// TIA Portal project "ConectaTwo" (V16)

(* hardware
DEVICE "S71500/ET200MP station_1"  S7-1500 station
   slot 0: "Rail_0"  Rack  6ES7 590-1***0-0AA0
   slot 1: "PLC_1"  CPU 1516-3 PN/DP  6ES7 516-3AN00-0AB0  V1.8
      slot 3: "CPU display_1"  6ES7591-1BA00-0AA0
      slot 32768: "PROFINET interface_1"  X1
         slot 32769: "Port_1"  X1 P1
         slot 32770: "Port_2"  X1 P2
      slot 33024: "PROFINET interface_2"  X2
         slot 33025: "Port_1"  X2 P1
      slot 33280: "DP interface_1"  X3
DEVICE "S71500/ET200MP station_2"  S7-1500 station
   slot 0: "Rail_0"  Rack  6ES7 590-1***0-0AA0
   slot 1: "PLC_2"  CPU 1516-3 PN/DP  6ES7 516-3AN00-0AB0  V1.8
      slot 3: "CPU display_1"  6ES7591-1BA00-0AA0
      slot 32768: "PROFINET interface_1"  X1
         slot 32769: "Port_1"  X1 P1
         slot 32770: "Port_2"  X1 P2
      slot 33024: "PROFINET interface_2"  X2
         slot 33025: "Port_1"  X2 P1
      slot 33280: "DP interface_1"  X3
DEVICE "HMI_1"  TP700 Comfort
   slot 0: "HMI_1"  TP700 Comfort  6AV2 124-0GC01-0AX0  16.0.0.0
   slot 1: "HMI_RT_1"  TP700 Comfort  6AV2 124-0GC01-0AX0  16.0.0.0
   slot 5: "HMI_1.IE_CP_1"  PROFINET Interface  16.0.0.0
      slot 1: "PROFINET Interface_1"  PROFINET Interface
         slot 1: "Port_1"  Port
         slot 2: "Port_2"  Port
   slot 7: "HMI_1.MPI/DP_CP_1"  MPI/DP Interface  16.0.0.0
DEVICE "HMI_2"  TP700 Comfort
   slot 0: "HMI_2"  TP700 Comfort  6AV2 124-0GC01-0AX0  16.0.0.0
   slot 1: "HMI_RT_2"  TP700 Comfort  6AV2 124-0GC01-0AX0  16.0.0.0
   slot 5: "HMI_2.IE_CP_1"  PROFINET Interface  16.0.0.0
      slot 1: "PROFINET Interface_1"  PROFINET Interface
         slot 1: "Port_1"  Port
         slot 2: "Port_2"  Port
   slot 7: "HMI_2.MPI/DP_CP_1"  MPI/DP Interface  16.0.0.0
*)

// ===== PLC "PLC_1"  CPU 1516-3 PN/DP =====

VAR_GLOBAL   // PLC tag table "Default tag table"
   "Clock_Byte" AT %MB10 : Byte;
   "Clock_10Hz" AT %M10.0 : Bool;
   "Clock_1Hz" AT %M10.5 : Bool;
   "Mensaje1J1" AT %M11.0 : Bool;
   "Mensaje2J1" AT %M11.1 : Bool;
   "Mensaje3J1" AT %M11.2 : Bool;
   "Mensaje4J1" AT %M11.3 : Bool;
   "Mensaje5J1" AT %M11.4 : Bool;
   "Mensaje6J1" AT %M11.5 : Bool;
   "Mensaje7J1" AT %M11.6 : Bool;
   "B1J1" AT %M11.7 : Bool;
   "B2J1" AT %M12.0 : Bool;
   "B3J1" AT %M12.1 : Bool;
   "B4J1" AT %M12.2 : Bool;
   "B5J1" AT %M12.3 : Bool;
   "B6J1" AT %M12.4 : Bool;
   "B7J1" AT %M12.5 : Bool;
   "B8J1" AT %M12.6 : Bool;
   "B9J1" AT %M12.7 : Bool;
   "PanelJ1" AT %M13.0 : Bool;
   "ReiniciarJ1" AT %M13.1 : Bool;
   "Conecta4J1" AT %M13.2 : Bool;
   "Conecta5J1" AT %M13.3 : Bool;
   "Conecta4SJ1" AT %M13.4 : Bool;
   "Conecta5SJ1" AT %M13.5 : Bool;
   "ModoJuegoJ1Send" AT %MW14 : Int;
   "ModoJuegoJ2Rec" AT %MW16 : Int;
   "ResetJ1Send" AT %M18.0 : Bool;
   "ResetJ2Rec" AT %M18.1 : Bool;
   "EstadoTurnoAJ1Send" AT %M18.2 : Bool;
   "EstadoTurnoAJ2Rec" AT %M18.3 : Bool;
   "EstadoTurnoBJ1Send" AT %M18.4 : Bool;
   "EstadoTurnoBJ2Rec" AT %M18.5 : Bool;
   "CambioBJ1" AT %M18.6 : Bool;
   "CambioVectorJ1" AT %M18.7 : Bool;
END_VAR

DATA_BLOCK "Jugador1Vect"   // DB4
{ S7_Optimized_Access := 'FALSE' }
VERSION : 0.1
   VAR
      J1Vect : Array[0..7, 0..8] of Int;
      J1VecSend : Array[0..7, 0..8] of Int;
      J1VecRec : Array[0..7, 0..8] of Int;
   END_VAR
BEGIN
   J1Vect[0,0] := 0;
   J1Vect[0,1] := 0;
   J1Vect[0,2] := 0;
   J1Vect[0,3] := 0;
   J1Vect[0,4] := 0;
   J1Vect[0,6] := 0;
   J1Vect[0,7] := 0;
   J1Vect[0,8] := 0;
   J1Vect[1,0] := 0;
   J1Vect[1,1] := 0;
   J1Vect[1,3] := 0;
   J1VecSend[1,3] := 0;
   J1VecSend[1,1] := 0;
   J1VecSend[1,0] := 0;
   J1VecSend[0,8] := 0;
   J1VecSend[0,7] := 0;
   J1VecSend[0,6] := 0;
   J1VecSend[0,4] := 0;
   J1VecSend[0,3] := 0;
   J1VecSend[0,2] := 0;
   J1VecSend[0,1] := 0;
   J1VecSend[0,0] := 0;
   J1VecRec[0,0] := 0;
   J1VecRec[0,1] := 0;
   J1VecRec[0,2] := 0;
   J1VecRec[0,3] := 0;
   J1VecRec[0,4] := 0;
   J1VecRec[0,6] := 0;
   J1VecRec[0,7] := 0;
   J1VecRec[0,8] := 0;
   J1VecRec[1,0] := 0;
   J1VecRec[1,1] := 0;
   J1VecRec[1,3] := 0;
END_DATA_BLOCK

// folder: System blocks/Program resources

DATA_BLOCK "EnviarModo"   // DB3
{ S7_Optimized_Access := 'TRUE' }
AUTHOR : SIMATIC
FAMILY : MC7Plus
NAME : TC_IP_v4
VERSION : 1.0
// stored: InstanceOfName TCON_IP_v4
"TCON_IP_v4"
BEGIN
   ID := 1;
   InterfaceId := 64;
   RemotePort := 2000;
   ActiveEstablished := true;
   RemoteAddress.ADDR[1] := 192;
   RemoteAddress.ADDR[2] := 168;
   RemoteAddress.ADDR[3] := 50;
   RemoteAddress.ADDR[4] := 2;
END_DATA_BLOCK

DATA_BLOCK "EnviarReset"   // DB6
{ S7_Optimized_Access := 'TRUE' }
AUTHOR : SIMATIC
FAMILY : MC7Plus
NAME : TC_IP_v4
VERSION : 1.0
// stored: InstanceOfName TCON_IP_v4
"TCON_IP_v4"
BEGIN
   ID := 2;
   InterfaceId := 64;
   RemotePort := 2010;
   ActiveEstablished := true;
   RemoteAddress.ADDR[1] := 192;
   RemoteAddress.ADDR[2] := 168;
   RemoteAddress.ADDR[3] := 50;
   RemoteAddress.ADDR[4] := 2;
END_DATA_BLOCK

DATA_BLOCK "EnviarTurnoA"   // DB7
{ S7_Optimized_Access := 'TRUE' }
AUTHOR : SIMATIC
FAMILY : MC7Plus
NAME : TC_IP_v4
VERSION : 1.0
// stored: InstanceOfName TCON_IP_v4
"TCON_IP_v4"
BEGIN
   ID := 3;
   InterfaceId := 64;
   RemotePort := 2020;
   ActiveEstablished := true;
   RemoteAddress.ADDR[1] := 192;
   RemoteAddress.ADDR[2] := 168;
   RemoteAddress.ADDR[3] := 50;
   RemoteAddress.ADDR[4] := 2;
END_DATA_BLOCK

DATA_BLOCK "RecibirTurnoB"   // DB9
{ S7_Optimized_Access := 'TRUE' }
AUTHOR : SIMATIC
FAMILY : MC7Plus
NAME : TC_IP_v4
VERSION : 1.0
// stored: InstanceOfName TCON_IP_v4
"TCON_IP_v4"
BEGIN
   ID := 4;
   InterfaceId := 64;
   LocalPort := 2030;
   RemoteAddress.ADDR[1] := 192;
   RemoteAddress.ADDR[2] := 168;
   RemoteAddress.ADDR[3] := 50;
   RemoteAddress.ADDR[4] := 2;
END_DATA_BLOCK

DATA_BLOCK "EnviarVectorA"   // DB12
{ S7_Optimized_Access := 'TRUE' }
AUTHOR : SIMATIC
FAMILY : MC7Plus
NAME : TC_IP_v4
VERSION : 1.0
// stored: InstanceOfName TCON_IP_v4
"TCON_IP_v4"
BEGIN
   ID := 5;
   InterfaceId := 64;
   RemotePort := 2040;
   ActiveEstablished := true;
   RemoteAddress.ADDR[1] := 192;
   RemoteAddress.ADDR[2] := 168;
   RemoteAddress.ADDR[3] := 50;
   RemoteAddress.ADDR[4] := 2;
END_DATA_BLOCK

DATA_BLOCK "RecibirVectorB"   // DB13
{ S7_Optimized_Access := 'TRUE' }
AUTHOR : SIMATIC
FAMILY : MC7Plus
NAME : TC_IP_v4
VERSION : 1.0
// stored: InstanceOfName TCON_IP_v4
"TCON_IP_v4"
BEGIN
   ID := 6;
   InterfaceId := 64;
   LocalPort := 2050;
   RemoteAddress.ADDR[1] := 192;
   RemoteAddress.ADDR[2] := 168;
   RemoteAddress.ADDR[3] := 50;
   RemoteAddress.ADDR[4] := 2;
END_DATA_BLOCK

// folder: (top level)

ORGANIZATION_BLOCK "Main"   // OB1, LAD, ProgramCycle
TITLE = "Main Program Sweep (Cycle)"
{ S7_Optimized_Access := 'TRUE' }
VERSION : 0.1
   VAR_INPUT
      Initial_Call : Bool;   // Initial call of this OB
      Remanence : Bool;   // =True, if remanent data are available
   END_VAR
BEGIN

REGION Network 1: Enviar y Recibir Modo de Juego
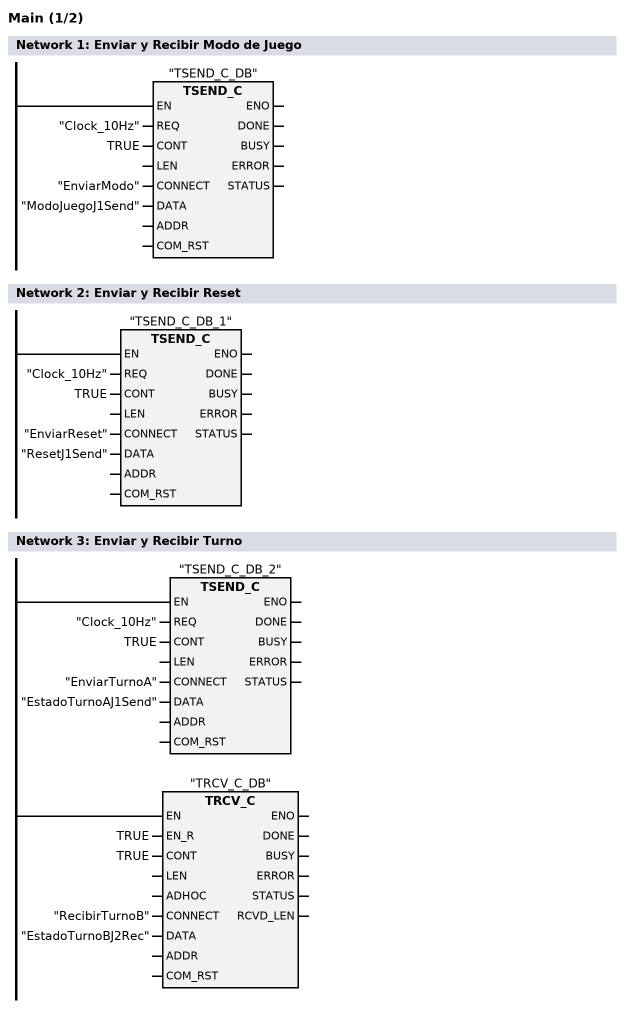
   "TSEND_C_DB"(REQ := "Clock_10Hz", CONT := TRUE, CONNECT := "EnviarModo", DATA := "ModoJuegoJ1Send");   // TSEND_C
END_REGION

REGION Network 2: Enviar y Recibir Reset
   "TSEND_C_DB_1"(REQ := "Clock_10Hz", CONT := TRUE, CONNECT := "EnviarReset", DATA := "ResetJ1Send");   // TSEND_C
END_REGION

REGION Network 3: Enviar y Recibir Turno
   "TSEND_C_DB_2"(REQ := "Clock_10Hz", CONT := TRUE, CONNECT := "EnviarTurnoA", DATA := "EstadoTurnoAJ1Send");   // TSEND_C
   "TRCV_C_DB"(EN_R := TRUE, CONT := TRUE, CONNECT := "RecibirTurnoB", DATA := "EstadoTurnoBJ2Rec");   // TRCV_C
END_REGION

REGION Network 4: Enviar y Recibir Vector
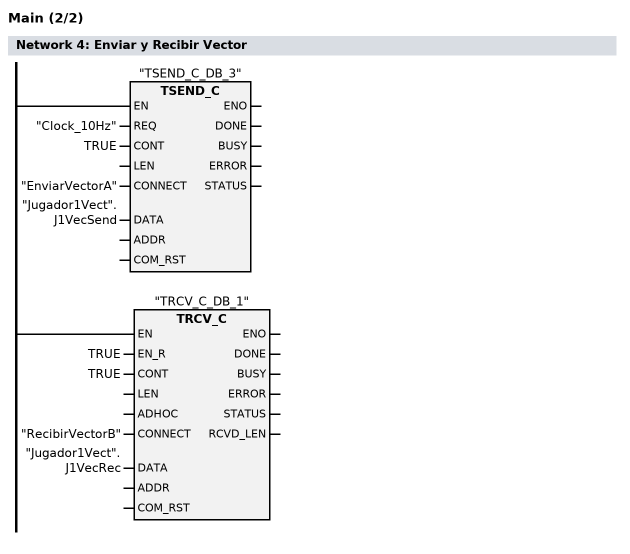
   "TSEND_C_DB_3"(REQ := "Clock_10Hz",   // TSEND_C
                  CONT := TRUE,
                  CONNECT := "EnviarVectorA",
                  DATA := "Jugador1Vect".J1VecSend);
   "TRCV_C_DB_1"(EN_R := TRUE, CONT := TRUE, CONNECT := "RecibirVectorB", DATA := "Jugador1Vect".J1VecRec);   // TRCV_C
END_REGION

REGION Network 5 (SCL): Checar si ganador rojo
   IF "ReiniciarJ1" = TRUE THEN
       "ResetJ1Send" := TRUE;
       "ModoJuegoJ1Send" := 0;
       "ModoJuegoJ2Rec" := 0;
       FILL_BLK(IN:=0,
                COUNT:=72,
                OUT=>"Jugador1Vect".J1Vect[0,0]);
       FILL_BLK(IN := 0,
                COUNT := 72,
                OUT => "Jugador1Vect".J1VecSend[0, 0]);
       FILL_BLK(IN := 0,
                COUNT := 72,
                OUT => "Jugador1Vect".J1VecRec[0, 0]);
       "Mensaje1J1" := FALSE;
       "Mensaje2J1" := FALSE;
       "Mensaje3J1" := FALSE;
       "Mensaje4J1" := FALSE;
       "Mensaje5J1" := FALSE;
       "Mensaje6J1" := FALSE;
       "Mensaje7J1" := FALSE;
       "EstadoTurnoAJ1Send" := TRUE;
       "EstadoTurnoAJ2Rec" := FALSE;
       "EstadoTurnoBJ1Send" := FALSE;
       "EstadoTurnoBJ2Rec" := FALSE;
       "Conecta4SJ1" := FALSE;
       "Conecta5SJ1" := FALSE;
       "PanelJ1" := FALSE;
       "CambioBJ1" := FALSE;
       "CambioVectorJ1" := FALSE;
   ELSE
       "ResetJ1Send" := FALSE;
   END_IF;

   IF "ModoJuegoJ1Send" = 0 THEN
       IF "Conecta4J1" = TRUE THEN
           "Conecta4SJ1" := TRUE;
           "ModoJuegoJ1Send" := 4;
           "Mensaje1J1" := TRUE;
           "Mensaje2J1" := TRUE;
           "Mensaje3J1" := FALSE;
       END_IF;
       IF "Conecta5J1" = TRUE THEN
           "Conecta5SJ1" := TRUE;
           "ModoJuegoJ1Send" := 5;
           "Mensaje1J1" := TRUE;
           "Mensaje3J1" := TRUE;
           "Mensaje2J1" := FALSE;
       END_IF;
   END_IF;

   IF "Conecta4SJ1" = TRUE OR "Conecta5SJ1" = TRUE THEN
       IF "EstadoTurnoAJ1Send" = TRUE THEN
           "PanelJ1" := TRUE;
           "Mensaje4J1" := TRUE;
           "Mensaje5J1" := FALSE;
       ELSE
           "PanelJ1" := FALSE;
           "Mensaje4J1" := FALSE;
           "Mensaje5J1" := TRUE;
       END_IF;
   END_IF;

   IF "B1J1" OR "B2J1" OR "B3J1" OR "B4J1" OR "B5J1" OR "B6J1" OR "B7J1" OR "B7J1" OR "B8J1" OR "B9J1" OR "EstadoTurnoBJ2Rec" THEN
       IF "EstadoTurnoAJ1Send" = TRUE THEN
           "EstadoTurnoAJ1Send" := FALSE;
       ELSE
           "EstadoTurnoAJ1Send" := TRUE;
       END_IF;
   END_IF;

   IF "B1J1" AND "CambioBJ1" = FALSE THEN
       MOVE_BLK(IN := "Jugador1Vect".J1VecRec[0, 0],
                COUNT := 72,
                OUT => "Jugador1Vect".J1Vect[0, 0]);
       IF "Jugador1Vect".J1Vect[0, 0] = 0 THEN
           "Jugador1Vect".J1Vect[0, 0] := 2;
           "CambioBJ1" := TRUE;
           MOVE_BLK(IN := "Jugador1Vect".J1Vect[0, 0],
                    COUNT := 72,
                    OUT => "Jugador1Vect".J1VecSend[0, 0]);
       ELSIF "Jugador1Vect".J1Vect[1, 0] = 0 THEN
           "Jugador1Vect".J1Vect[1, 0] := 2;
           "CambioBJ1" := TRUE;
           MOVE_BLK(IN := "Jugador1Vect".J1VecRec[0, 0],
                    COUNT := 72,
                    OUT => "Jugador1Vect".J1Vect[0, 0]);
       ELSIF "Jugador1Vect".J1Vect[2, 0] = 0 THEN
           "Jugador1Vect".J1Vect[2, 0] := 2;
           "CambioBJ1" := TRUE;
           MOVE_BLK(IN := "Jugador1Vect".J1Vect[0, 0],
                    COUNT := 72,
                    OUT => "Jugador1Vect".J1VecSend[0, 0]);
       ELSIF "Jugador1Vect".J1Vect[3, 0] = 0 THEN
           "Jugador1Vect".J1Vect[3, 0] := 2;
           "CambioBJ1" := TRUE;
           MOVE_BLK(IN := "Jugador1Vect".J1VecRec[0, 0],
                    COUNT := 72,
                    OUT => "Jugador1Vect".J1Vect[0, 0]);
       ELSIF "Jugador1Vect".J1Vect[4, 0] = 0 THEN
           "Jugador1Vect".J1Vect[4, 0] := 2;
           "CambioBJ1" := TRUE;
           MOVE_BLK(IN := "Jugador1Vect".J1Vect[0, 0],
                    COUNT := 72,
                    OUT => "Jugador1Vect".J1VecSend[0, 0]);
       ELSIF "Jugador1Vect".J1Vect[5, 0] = 0 THEN
           "Jugador1Vect".J1Vect[5, 0] := 2;
           "CambioBJ1" := TRUE;
           MOVE_BLK(IN := "Jugador1Vect".J1Vect[0, 0],
                    COUNT := 72,
                    OUT => "Jugador1Vect".J1VecSend[0, 0]);
       ELSIF "Jugador1Vect".J1Vect[6, 0] = 0 THEN
           "Jugador1Vect".J1Vect[6, 0] := 2;
           "CambioBJ1" := TRUE;
           MOVE_BLK(IN := "Jugador1Vect".J1Vect[0, 0],
                    COUNT := 72,
                    OUT => "Jugador1Vect".J1VecSend[0, 0]);
       ELSIF "Jugador1Vect".J1Vect[7, 0] = 0 THEN
           "Jugador1Vect".J1Vect[7, 0] := 2;
           "CambioBJ1" := TRUE;
           MOVE_BLK(IN := "Jugador1Vect".J1Vect[0, 0],
                    COUNT := 72,
                    OUT => "Jugador1Vect".J1VecSend[0, 0]);
       END_IF;
   END_IF;

   IF "B2J1" AND "CambioBJ1" = FALSE THEN
       MOVE_BLK(IN := "Jugador1Vect".J1VecRec[0, 0],
                COUNT := 72,
                OUT => "Jugador1Vect".J1Vect[0, 0]);
       IF "Jugador1Vect".J1Vect[0, 1] = 0 THEN
           "Jugador1Vect".J1Vect[0, 1] := 2;
           "CambioBJ1" := TRUE;
           MOVE_BLK(IN := "Jugador1Vect".J1Vect[0, 0],
                    COUNT := 72,
                    OUT => "Jugador1Vect".J1VecSend[0, 0]);
       ELSIF "Jugador1Vect".J1Vect[1, 1] = 0 THEN
           "Jugador1Vect".J1Vect[1, 1] := 2;
           "CambioBJ1" := TRUE;
           MOVE_BLK(IN := "Jugador1Vect".J1VecRec[0, 0],
                    COUNT := 72,
                    OUT => "Jugador1Vect".J1Vect[0, 0]);
       ELSIF "Jugador1Vect".J1Vect[2, 1] = 0 THEN
           "Jugador1Vect".J1Vect[2, 1] := 2;
           "CambioBJ1" := TRUE;
           MOVE_BLK(IN := "Jugador1Vect".J1Vect[0, 0],
                    COUNT := 72,
                    OUT => "Jugador1Vect".J1VecSend[0, 0]);
       ELSIF "Jugador1Vect".J1Vect[3, 1] = 0 THEN
           "Jugador1Vect".J1Vect[3, 1] := 2;
           "CambioBJ1" := TRUE;
           MOVE_BLK(IN := "Jugador1Vect".J1VecRec[0, 0],
                    COUNT := 72,
                    OUT => "Jugador1Vect".J1Vect[0, 0]);
       ELSIF "Jugador1Vect".J1Vect[4, 1] = 0 THEN
           "Jugador1Vect".J1Vect[4, 1] := 2;
           "CambioBJ1" := TRUE;
           MOVE_BLK(IN := "Jugador1Vect".J1Vect[0, 0],
                    COUNT := 72,
                    OUT => "Jugador1Vect".J1VecSend[0, 0]);
       ELSIF "Jugador1Vect".J1Vect[5, 1] = 0 THEN
           "Jugador1Vect".J1Vect[5, 1] := 2;
           "CambioBJ1" := TRUE;
           MOVE_BLK(IN := "Jugador1Vect".J1Vect[0, 0],
                    COUNT := 72,
                    OUT => "Jugador1Vect".J1VecSend[0, 0]);
       ELSIF "Jugador1Vect".J1Vect[6, 1] = 0 THEN
           "Jugador1Vect".J1Vect[6, 1] := 2;
           "CambioBJ1" := TRUE;
           MOVE_BLK(IN := "Jugador1Vect".J1Vect[0, 0],
                    COUNT := 72,
                    OUT => "Jugador1Vect".J1VecSend[0, 0]);
       ELSIF "Jugador1Vect".J1Vect[7, 1] = 0 THEN
           "Jugador1Vect".J1Vect[7, 1] := 2;
           "CambioBJ1" := TRUE;
           MOVE_BLK(IN := "Jugador1Vect".J1Vect[0, 0],
                    COUNT := 72,
                    OUT => "Jugador1Vect".J1VecSend[0, 0]);
       END_IF;
   END_IF;

   IF "B3J1" AND "CambioBJ1" = FALSE THEN
       MOVE_BLK(IN := "Jugador1Vect".J1VecRec[0, 0],
                COUNT := 72,
                OUT => "Jugador1Vect".J1Vect[0, 0]);
       IF "Jugador1Vect".J1Vect[0, 2] = 0 THEN
           "Jugador1Vect".J1Vect[0, 2] := 2;
           "CambioBJ1" := TRUE;
           MOVE_BLK(IN := "Jugador1Vect".J1Vect[0, 0],
                    COUNT := 72,
                    OUT => "Jugador1Vect".J1VecSend[0, 0]);
       ELSIF "Jugador1Vect".J1Vect[1, 2] = 0 THEN
           "Jugador1Vect".J1Vect[1, 2] := 2;
           "CambioBJ1" := TRUE;
           MOVE_BLK(IN := "Jugador1Vect".J1VecRec[0, 0],
                    COUNT := 72,
                    OUT => "Jugador1Vect".J1Vect[0, 0]);
       ELSIF "Jugador1Vect".J1Vect[2, 2] = 0 THEN
           "Jugador1Vect".J1Vect[2, 2] := 2;
           "CambioBJ1" := TRUE;
           MOVE_BLK(IN := "Jugador1Vect".J1Vect[0, 0],
                    COUNT := 72,
                    OUT => "Jugador1Vect".J1VecSend[0, 0]);
       ELSIF "Jugador1Vect".J1Vect[3, 2] = 0 THEN
           "Jugador1Vect".J1Vect[3, 2] := 2;
           "CambioBJ1" := TRUE;
           MOVE_BLK(IN := "Jugador1Vect".J1VecRec[0, 0],
                    COUNT := 72,
                    OUT => "Jugador1Vect".J1Vect[0, 0]);
       ELSIF "Jugador1Vect".J1Vect[4, 2] = 0 THEN
           "Jugador1Vect".J1Vect[4, 2] := 2;
           "CambioBJ1" := TRUE;
           MOVE_BLK(IN := "Jugador1Vect".J1Vect[0, 0],
                    COUNT := 72,
                    OUT => "Jugador1Vect".J1VecSend[0, 0]);
       ELSIF "Jugador1Vect".J1Vect[5, 2] = 0 THEN
           "Jugador1Vect".J1Vect[5, 2] := 2;
           "CambioBJ1" := TRUE;
           MOVE_BLK(IN := "Jugador1Vect".J1Vect[0, 0],
                    COUNT := 72,
                    OUT => "Jugador1Vect".J1VecSend[0, 0]);
       ELSIF "Jugador1Vect".J1Vect[6, 2] = 0 THEN
           "Jugador1Vect".J1Vect[6, 2] := 2;
           "CambioBJ1" := TRUE;
           MOVE_BLK(IN := "Jugador1Vect".J1Vect[0, 0],
                    COUNT := 72,
                    OUT => "Jugador1Vect".J1VecSend[0, 0]);
       ELSIF "Jugador1Vect".J1Vect[7, 2] = 0 THEN
           "Jugador1Vect".J1Vect[7, 2] := 2;
           "CambioBJ1" := TRUE;
           MOVE_BLK(IN := "Jugador1Vect".J1Vect[0, 0],
                    COUNT := 72,
                    OUT => "Jugador1Vect".J1VecSend[0, 0]);
       END_IF;
   END_IF;

   IF "B4J1" AND "CambioBJ1" = FALSE THEN
       MOVE_BLK(IN := "Jugador1Vect".J1VecRec[0, 0],
                COUNT := 72,
                OUT => "Jugador1Vect".J1Vect[0, 0]);
       IF "Jugador1Vect".J1Vect[0, 3] = 0 THEN
           "Jugador1Vect".J1Vect[0, 3] := 2;
           "CambioBJ1" := TRUE;
           MOVE_BLK(IN := "Jugador1Vect".J1Vect[0, 0],
                    COUNT := 72,
                    OUT => "Jugador1Vect".J1VecSend[0, 0]);
       ELSIF "Jugador1Vect".J1Vect[1, 3] = 0 THEN
           "Jugador1Vect".J1Vect[1, 3] := 2;
           "CambioBJ1" := TRUE;
           MOVE_BLK(IN := "Jugador1Vect".J1VecRec[0, 0],
                    COUNT := 72,
                    OUT => "Jugador1Vect".J1Vect[0, 0]);
       ELSIF "Jugador1Vect".J1Vect[2, 3] = 0 THEN
           "Jugador1Vect".J1Vect[2, 3] := 2;
           "CambioBJ1" := TRUE;
           MOVE_BLK(IN := "Jugador1Vect".J1Vect[0, 0],
                    COUNT := 72,
                    OUT => "Jugador1Vect".J1VecSend[0, 0]);
       ELSIF "Jugador1Vect".J1Vect[3, 3] = 0 THEN
           "Jugador1Vect".J1Vect[3, 3] := 2;
           "CambioBJ1" := TRUE;
           MOVE_BLK(IN := "Jugador1Vect".J1VecRec[0, 0],
                    COUNT := 72,
                    OUT => "Jugador1Vect".J1Vect[0, 0]);
       ELSIF "Jugador1Vect".J1Vect[4, 3] = 0 THEN
           "Jugador1Vect".J1Vect[4, 3] := 2;
           "CambioBJ1" := TRUE;
           MOVE_BLK(IN := "Jugador1Vect".J1Vect[0, 0],
                    COUNT := 72,
                    OUT => "Jugador1Vect".J1VecSend[0, 0]);
       ELSIF "Jugador1Vect".J1Vect[5, 3] = 0 THEN
           "Jugador1Vect".J1Vect[5, 3] := 2;
           "CambioBJ1" := TRUE;
           MOVE_BLK(IN := "Jugador1Vect".J1Vect[0, 0],
                    COUNT := 72,
                    OUT => "Jugador1Vect".J1VecSend[0, 0]);
       ELSIF "Jugador1Vect".J1Vect[6, 3] = 0 THEN
           "Jugador1Vect".J1Vect[6, 3] := 2;
           "CambioBJ1" := TRUE;
           MOVE_BLK(IN := "Jugador1Vect".J1Vect[0, 0],
                    COUNT := 72,
                    OUT => "Jugador1Vect".J1VecSend[0, 0]);
       ELSIF "Jugador1Vect".J1Vect[7, 3] = 0 THEN
           "Jugador1Vect".J1Vect[7, 3] := 2;
           "CambioBJ1" := TRUE;
           MOVE_BLK(IN := "Jugador1Vect".J1Vect[0, 0],
                    COUNT := 72,
                    OUT => "Jugador1Vect".J1VecSend[0, 0]);
       END_IF;
   END_IF;

   IF "B5J1" AND "CambioBJ1" = FALSE THEN
       MOVE_BLK(IN := "Jugador1Vect".J1VecRec[0, 0],
                COUNT := 72,
                OUT => "Jugador1Vect".J1Vect[0, 0]);
       IF "Jugador1Vect".J1Vect[0, 4] = 0 THEN
           "Jugador1Vect".J1Vect[0, 4] := 2;
           "CambioBJ1" := TRUE;
           MOVE_BLK(IN := "Jugador1Vect".J1Vect[0, 0],
                    COUNT := 72,
                    OUT => "Jugador1Vect".J1VecSend[0, 0]);
       ELSIF "Jugador1Vect".J1Vect[1, 4] = 0 THEN
           "Jugador1Vect".J1Vect[1, 4] := 2;
           "CambioBJ1" := TRUE;
           MOVE_BLK(IN := "Jugador1Vect".J1VecRec[0, 0],
                    COUNT := 72,
                    OUT => "Jugador1Vect".J1Vect[0, 0]);
       ELSIF "Jugador1Vect".J1Vect[2, 4] = 0 THEN
           "Jugador1Vect".J1Vect[2, 4] := 2;
           "CambioBJ1" := TRUE;
           MOVE_BLK(IN := "Jugador1Vect".J1Vect[0, 0],
                    COUNT := 72,
                    OUT => "Jugador1Vect".J1VecSend[0, 0]);
       ELSIF "Jugador1Vect".J1Vect[3, 4] = 0 THEN
           "Jugador1Vect".J1Vect[3, 4] := 2;
           "CambioBJ1" := TRUE;
           MOVE_BLK(IN := "Jugador1Vect".J1VecRec[0, 0],
                    COUNT := 72,
                    OUT => "Jugador1Vect".J1Vect[0, 0]);
       ELSIF "Jugador1Vect".J1Vect[4, 4] = 0 THEN
           "Jugador1Vect".J1Vect[4, 4] := 2;
           "CambioBJ1" := TRUE;
           MOVE_BLK(IN := "Jugador1Vect".J1Vect[0, 0],
                    COUNT := 72,
                    OUT => "Jugador1Vect".J1VecSend[0, 0]);
       ELSIF "Jugador1Vect".J1Vect[5, 4] = 0 THEN
           "Jugador1Vect".J1Vect[5, 4] := 2;
           "CambioBJ1" := TRUE;
           MOVE_BLK(IN := "Jugador1Vect".J1Vect[0, 0],
                    COUNT := 72,
                    OUT => "Jugador1Vect".J1VecSend[0, 0]);
       ELSIF "Jugador1Vect".J1Vect[6, 4] = 0 THEN
           "Jugador1Vect".J1Vect[6, 4] := 2;
           "CambioBJ1" := TRUE;
           MOVE_BLK(IN := "Jugador1Vect".J1Vect[0, 0],
                    COUNT := 72,
                    OUT => "Jugador1Vect".J1VecSend[0, 0]);
       ELSIF "Jugador1Vect".J1Vect[7, 4] = 0 THEN
           "Jugador1Vect".J1Vect[7, 4] := 2;
           "CambioBJ1" := TRUE;
           MOVE_BLK(IN := "Jugador1Vect".J1Vect[0, 0],
                    COUNT := 72,
                    OUT => "Jugador1Vect".J1VecSend[0, 0]);
       END_IF;
   END_IF;

   IF "B6J1" AND "CambioBJ1" = FALSE THEN
       MOVE_BLK(IN := "Jugador1Vect".J1VecRec[0, 0],
                COUNT := 72,
                OUT => "Jugador1Vect".J1Vect[0, 0]);
       IF "Jugador1Vect".J1Vect[0, 5] = 0 THEN
           "Jugador1Vect".J1Vect[0, 5] := 2;
           "CambioBJ1" := TRUE;
           MOVE_BLK(IN := "Jugador1Vect".J1Vect[0, 0],
                    COUNT := 72,
                    OUT => "Jugador1Vect".J1VecSend[0, 0]);
       ELSIF "Jugador1Vect".J1Vect[1, 5] = 0 THEN
           "Jugador1Vect".J1Vect[1, 5] := 2;
           "CambioBJ1" := TRUE;
           MOVE_BLK(IN := "Jugador1Vect".J1VecRec[0, 0],
                    COUNT := 72,
                    OUT => "Jugador1Vect".J1Vect[0, 0]);
       ELSIF "Jugador1Vect".J1Vect[2, 5] = 0 THEN
           "Jugador1Vect".J1Vect[2, 5] := 2;
           "CambioBJ1" := TRUE;
           MOVE_BLK(IN := "Jugador1Vect".J1Vect[0, 0],
                    COUNT := 72,
                    OUT => "Jugador1Vect".J1VecSend[0, 0]);
       ELSIF "Jugador1Vect".J1Vect[3, 5] = 0 THEN
           "Jugador1Vect".J1Vect[3, 5] := 2;
           "CambioBJ1" := TRUE;
           MOVE_BLK(IN := "Jugador1Vect".J1VecRec[0, 0],
                    COUNT := 72,
                    OUT => "Jugador1Vect".J1Vect[0, 0]);
       ELSIF "Jugador1Vect".J1Vect[4, 5] = 0 THEN
           "Jugador1Vect".J1Vect[4, 5] := 2;
           "CambioBJ1" := TRUE;
           MOVE_BLK(IN := "Jugador1Vect".J1Vect[0, 0],
                    COUNT := 72,
                    OUT => "Jugador1Vect".J1VecSend[0, 0]);
       ELSIF "Jugador1Vect".J1Vect[5, 5] = 0 THEN
           "Jugador1Vect".J1Vect[5, 5] := 2;
           "CambioBJ1" := TRUE;
           MOVE_BLK(IN := "Jugador1Vect".J1Vect[0, 0],
                    COUNT := 72,
                    OUT => "Jugador1Vect".J1VecSend[0, 0]);
       ELSIF "Jugador1Vect".J1Vect[6, 5] = 0 THEN
           "Jugador1Vect".J1Vect[6, 5] := 2;
           "CambioBJ1" := TRUE;
           MOVE_BLK(IN := "Jugador1Vect".J1Vect[0, 0],
                    COUNT := 72,
                    OUT => "Jugador1Vect".J1VecSend[0, 0]);
       ELSIF "Jugador1Vect".J1Vect[7, 5] = 0 THEN
           "Jugador1Vect".J1Vect[7, 5] := 2;
           "CambioBJ1" := TRUE;
           MOVE_BLK(IN := "Jugador1Vect".J1Vect[0, 0],
                    COUNT := 72,
                    OUT => "Jugador1Vect".J1VecSend[0, 0]);
       END_IF;
   END_IF;

   IF "B7J1" AND "CambioBJ1" = FALSE THEN
       MOVE_BLK(IN := "Jugador1Vect".J1VecRec[0, 0],
                COUNT := 72,
                OUT => "Jugador1Vect".J1Vect[0, 0]);
       IF "Jugador1Vect".J1Vect[0, 6] = 0 THEN
           "Jugador1Vect".J1Vect[0, 6] := 2;
           "CambioBJ1" := TRUE;
           MOVE_BLK(IN := "Jugador1Vect".J1Vect[0, 0],
                    COUNT := 72,
                    OUT => "Jugador1Vect".J1VecSend[0, 0]);
       ELSIF "Jugador1Vect".J1Vect[1, 6] = 0 THEN
           "Jugador1Vect".J1Vect[1, 6] := 2;
           "CambioBJ1" := TRUE;
           MOVE_BLK(IN := "Jugador1Vect".J1VecRec[0, 0],
                    COUNT := 72,
                    OUT => "Jugador1Vect".J1Vect[0, 0]);
       ELSIF "Jugador1Vect".J1Vect[2, 6] = 0 THEN
           "Jugador1Vect".J1Vect[2, 6] := 2;
           "CambioBJ1" := TRUE;
           MOVE_BLK(IN := "Jugador1Vect".J1Vect[0, 0],
                    COUNT := 72,
                    OUT => "Jugador1Vect".J1VecSend[0, 0]);
       ELSIF "Jugador1Vect".J1Vect[3, 6] = 0 THEN
           "Jugador1Vect".J1Vect[3, 6] := 2;
           "CambioBJ1" := TRUE;
           MOVE_BLK(IN := "Jugador1Vect".J1VecRec[0, 0],
                    COUNT := 72,
                    OUT => "Jugador1Vect".J1Vect[0, 0]);
       ELSIF "Jugador1Vect".J1Vect[4, 6] = 0 THEN
           "Jugador1Vect".J1Vect[4, 6] := 2;
           "CambioBJ1" := TRUE;
           MOVE_BLK(IN := "Jugador1Vect".J1Vect[0, 0],
                    COUNT := 72,
                    OUT => "Jugador1Vect".J1VecSend[0, 0]);
       ELSIF "Jugador1Vect".J1Vect[5, 6] = 0 THEN
           "Jugador1Vect".J1Vect[5, 6] := 2;
           "CambioBJ1" := TRUE;
           MOVE_BLK(IN := "Jugador1Vect".J1Vect[0, 0],
                    COUNT := 72,
                    OUT => "Jugador1Vect".J1VecSend[0, 0]);
       ELSIF "Jugador1Vect".J1Vect[6, 6] = 0 THEN
           "Jugador1Vect".J1Vect[6, 6] := 2;
           "CambioBJ1" := TRUE;
           MOVE_BLK(IN := "Jugador1Vect".J1Vect[0, 0],
                    COUNT := 72,
                    OUT => "Jugador1Vect".J1VecSend[0, 0]);
       ELSIF "Jugador1Vect".J1Vect[7, 6] = 0 THEN
           "Jugador1Vect".J1Vect[7, 6] := 2;
           "CambioBJ1" := TRUE;
           MOVE_BLK(IN := "Jugador1Vect".J1Vect[0, 0],
                    COUNT := 72,
                    OUT => "Jugador1Vect".J1VecSend[0, 0]);
       END_IF;
   END_IF;

   IF "B8J1" AND "CambioBJ1" = FALSE THEN
       MOVE_BLK(IN := "Jugador1Vect".J1VecRec[0, 0],
                COUNT := 72,
                OUT => "Jugador1Vect".J1Vect[0, 0]);
       IF "Jugador1Vect".J1Vect[0, 7] = 0 THEN
           "Jugador1Vect".J1Vect[0, 7] := 2;
           "CambioBJ1" := TRUE;
           MOVE_BLK(IN := "Jugador1Vect".J1Vect[0, 0],
                    COUNT := 72,
                    OUT => "Jugador1Vect".J1VecSend[0, 0]);
       ELSIF "Jugador1Vect".J1Vect[1, 7] = 0 THEN
           "Jugador1Vect".J1Vect[1, 7] := 2;
           "CambioBJ1" := TRUE;
           MOVE_BLK(IN := "Jugador1Vect".J1VecRec[0, 0],
                    COUNT := 72,
                    OUT => "Jugador1Vect".J1Vect[0, 0]);
       ELSIF "Jugador1Vect".J1Vect[2, 7] = 0 THEN
           "Jugador1Vect".J1Vect[2, 7] := 2;
           "CambioBJ1" := TRUE;
           MOVE_BLK(IN := "Jugador1Vect".J1Vect[0, 0],
                    COUNT := 72,
                    OUT => "Jugador1Vect".J1VecSend[0, 0]);
       ELSIF "Jugador1Vect".J1Vect[3, 7] = 0 THEN
           "Jugador1Vect".J1Vect[3, 7] := 2;
           "CambioBJ1" := TRUE;
           MOVE_BLK(IN := "Jugador1Vect".J1VecRec[0, 0],
                    COUNT := 72,
                    OUT => "Jugador1Vect".J1Vect[0, 0]);
       ELSIF "Jugador1Vect".J1Vect[4, 7] = 0 THEN
           "Jugador1Vect".J1Vect[4, 7] := 2;
           "CambioBJ1" := TRUE;
           MOVE_BLK(IN := "Jugador1Vect".J1Vect[0, 0],
                    COUNT := 72,
                    OUT => "Jugador1Vect".J1VecSend[0, 0]);
       ELSIF "Jugador1Vect".J1Vect[5, 7] = 0 THEN
           "Jugador1Vect".J1Vect[5, 7] := 2;
           "CambioBJ1" := TRUE;
           MOVE_BLK(IN := "Jugador1Vect".J1Vect[0, 0],
                    COUNT := 72,
                    OUT => "Jugador1Vect".J1VecSend[0, 0]);
       ELSIF "Jugador1Vect".J1Vect[6, 7] = 0 THEN
           "Jugador1Vect".J1Vect[6, 7] := 2;
           "CambioBJ1" := TRUE;
           MOVE_BLK(IN := "Jugador1Vect".J1Vect[0, 0],
                    COUNT := 72,
                    OUT => "Jugador1Vect".J1VecSend[0, 0]);
       ELSIF "Jugador1Vect".J1Vect[7, 7] = 0 THEN
           "Jugador1Vect".J1Vect[7, 7] := 2;
           "CambioBJ1" := TRUE;
           MOVE_BLK(IN := "Jugador1Vect".J1Vect[0, 0],
                    COUNT := 72,
                    OUT => "Jugador1Vect".J1VecSend[0, 0]);
       END_IF;
   END_IF;

   IF "B9J1" AND "CambioBJ1" = FALSE THEN
       MOVE_BLK(IN := "Jugador1Vect".J1VecRec[0, 0],
                COUNT := 72,
                OUT => "Jugador1Vect".J1Vect[0, 0]);
       IF "Jugador1Vect".J1Vect[0, 8] = 0 THEN
           "Jugador1Vect".J1Vect[0, 8] := 2;
           "CambioBJ1" := TRUE;
           MOVE_BLK(IN := "Jugador1Vect".J1Vect[0, 0],
                    COUNT := 72,
                    OUT => "Jugador1Vect".J1VecSend[0, 0]);
       ELSIF "Jugador1Vect".J1Vect[1, 8] = 0 THEN
           "Jugador1Vect".J1Vect[1, 8] := 2;
           "CambioBJ1" := TRUE;
           MOVE_BLK(IN := "Jugador1Vect".J1VecRec[0, 0],
                    COUNT := 72,
                    OUT => "Jugador1Vect".J1Vect[0, 0]);
       ELSIF "Jugador1Vect".J1Vect[2, 8] = 0 THEN
           "Jugador1Vect".J1Vect[2, 8] := 2;
           "CambioBJ1" := TRUE;
           MOVE_BLK(IN := "Jugador1Vect".J1Vect[0, 0],
                    COUNT := 72,
                    OUT => "Jugador1Vect".J1VecSend[0, 0]);
       ELSIF "Jugador1Vect".J1Vect[3, 8] = 0 THEN
           "Jugador1Vect".J1Vect[3, 8] := 2;
           "CambioBJ1" := TRUE;
           MOVE_BLK(IN := "Jugador1Vect".J1VecRec[0, 0],
                    COUNT := 72,
                    OUT => "Jugador1Vect".J1Vect[0, 0]);
       ELSIF "Jugador1Vect".J1Vect[4, 8] = 0 THEN
           "Jugador1Vect".J1Vect[4, 8] := 2;
           "CambioBJ1" := TRUE;
           MOVE_BLK(IN := "Jugador1Vect".J1Vect[0, 0],
                    COUNT := 72,
                    OUT => "Jugador1Vect".J1VecSend[0, 0]);
       ELSIF "Jugador1Vect".J1Vect[5, 8] = 0 THEN
           "Jugador1Vect".J1Vect[5, 8] := 2;
           "CambioBJ1" := TRUE;
           MOVE_BLK(IN := "Jugador1Vect".J1Vect[0, 0],
                    COUNT := 72,
                    OUT => "Jugador1Vect".J1VecSend[0, 0]);
       ELSIF "Jugador1Vect".J1Vect[6, 8] = 0 THEN
           "Jugador1Vect".J1Vect[6, 8] := 2;
           "CambioBJ1" := TRUE;
           MOVE_BLK(IN := "Jugador1Vect".J1Vect[0, 0],
                    COUNT := 72,
                    OUT => "Jugador1Vect".J1VecSend[0, 0]);
       ELSIF "Jugador1Vect".J1Vect[7, 8] = 0 THEN
           "Jugador1Vect".J1Vect[7, 8] := 2;
           "CambioBJ1" := TRUE;
           MOVE_BLK(IN := "Jugador1Vect".J1Vect[0, 0],
                    COUNT := 72,
                    OUT => "Jugador1Vect".J1VecSend[0, 0]);
       END_IF;
   END_IF;

   IF ("B1J1" = FALSE OR "B2J1" = FALSE OR "B3J1" = FALSE OR "B4J1" = FALSE OR "B5J1" = FALSE OR "B6J1" = FALSE OR "B7J1" = FALSE OR "B8J1" = FALSE OR "B9J1" = FALSE) AND "CambioBJ1" = TRUE THEN
       "CambioBJ1" := FALSE;
       "CambioVectorJ1" := FALSE;
   END_IF;
END_REGION
END_ORGANIZATION_BLOCK

// ===== PLC "PLC_2"  CPU 1516-3 PN/DP =====

VAR_GLOBAL   // PLC tag table "Default tag table"
   "Clock_Byte" AT %MB10 : Byte;
   "Clock_10Hz" AT %M10.0 : Bool;
   "Clock_1Hz" AT %M10.5 : Bool;
   "Mensaje1J2" AT %M11.0 : Bool;
   "Mensaje2J2" AT %M11.1 : Bool;
   "Mensaje3J2" AT %M11.2 : Bool;
   "Mensaje4J2" AT %M11.3 : Bool;
   "Mensaje5J2" AT %M11.4 : Bool;
   "Mensaje6J2" AT %M11.5 : Bool;
   "Mensaje7J2" AT %M11.6 : Bool;
   "B1J2" AT %M11.7 : Bool;
   "B2J2" AT %M12.0 : Bool;
   "B3J2" AT %M12.1 : Bool;
   "B4J2" AT %M12.2 : Bool;
   "B5J2" AT %M12.3 : Bool;
   "B6J2" AT %M12.4 : Bool;
   "B7J2" AT %M12.5 : Bool;
   "B8J2" AT %M12.6 : Bool;
   "B9J2" AT %M12.7 : Bool;
   "PanelJ2" AT %M13.0 : Bool;
   "ReiniciarJ2" AT %M13.1 : Bool;
   "Conecta4J2" AT %M13.2 : Bool;
   "Conecta5J2" AT %M13.3 : Bool;
   "Conecta4SJ2" AT %M13.4 : Bool;
   "Conecta5SJ2" AT %M13.5 : Bool;
   "ModoJuegoJ2Send" AT %MW14 : Int;
   "ModoJuegoJ1Rec" AT %MW16 : Int;
   "ResetJ2Send" AT %M18.0 : Bool;
   "ResetJ1Rec" AT %M18.1 : Bool;
   "EstadoTurnoAJ2Send" AT %M18.2 : Bool;
   "EstadoTurnoAJ1Rec" AT %M18.3 : Bool;
   "EstadoTurnoBJ2Send" AT %M18.4 : Bool;
   "EstadoTurnoBJ1Rec" AT %M18.5 : Bool;
   "CambioBJ2" AT %M18.7 : Bool;
   "CambioVectorJ2" AT %M19.0 : Bool;
END_VAR

DATA_BLOCK "Jugador2Vect"   // DB4
{ S7_Optimized_Access := 'FALSE' }
VERSION : 0.1
   VAR
      J2Vect : Array[0..7, 0..8] of Int;
      J2VecSend : Array[0..7, 0..8] of Int;
      J2VecRec : Array[0..7, 0..8] of Int;
   END_VAR
BEGIN
END_DATA_BLOCK

// folder: System blocks/Program resources

DATA_BLOCK "RecibirModo"   // DB5
{ S7_Optimized_Access := 'TRUE' }
AUTHOR : SIMATIC
FAMILY : MC7Plus
NAME : TC_IP_v4
VERSION : 1.0
// stored: InstanceOfName TCON_IP_v4
"TCON_IP_v4"
BEGIN
   ID := 1;
   InterfaceId := 64;
   LocalPort := 2000;
   RemoteAddress.ADDR[1] := 192;
   RemoteAddress.ADDR[2] := 168;
   RemoteAddress.ADDR[3] := 50;
   RemoteAddress.ADDR[4] := 1;
END_DATA_BLOCK

DATA_BLOCK "RecibirReset"   // DB6
{ S7_Optimized_Access := 'TRUE' }
AUTHOR : SIMATIC
FAMILY : MC7Plus
NAME : TC_IP_v4
VERSION : 1.0
// stored: InstanceOfName TCON_IP_v4
"TCON_IP_v4"
BEGIN
   ID := 2;
   InterfaceId := 64;
   LocalPort := 2010;
   RemoteAddress.ADDR[1] := 192;
   RemoteAddress.ADDR[2] := 168;
   RemoteAddress.ADDR[3] := 50;
   RemoteAddress.ADDR[4] := 1;
END_DATA_BLOCK

DATA_BLOCK "RecibirTurnoA"   // DB7
{ S7_Optimized_Access := 'TRUE' }
AUTHOR : SIMATIC
FAMILY : MC7Plus
NAME : TC_IP_v4
VERSION : 1.0
// stored: InstanceOfName TCON_IP_v4
"TCON_IP_v4"
BEGIN
   ID := 3;
   InterfaceId := 64;
   LocalPort := 2020;
   RemoteAddress.ADDR[1] := 192;
   RemoteAddress.ADDR[2] := 168;
   RemoteAddress.ADDR[3] := 50;
   RemoteAddress.ADDR[4] := 1;
END_DATA_BLOCK

DATA_BLOCK "EnviarTurnoB"   // DB8
{ S7_Optimized_Access := 'TRUE' }
AUTHOR : SIMATIC
FAMILY : MC7Plus
NAME : TC_IP_v4
VERSION : 1.0
// stored: InstanceOfName TCON_IP_v4
"TCON_IP_v4"
BEGIN
   ID := 4;
   InterfaceId := 64;
   RemotePort := 2030;
   ActiveEstablished := true;
   RemoteAddress.ADDR[1] := 192;
   RemoteAddress.ADDR[2] := 168;
   RemoteAddress.ADDR[3] := 50;
   RemoteAddress.ADDR[4] := 1;
END_DATA_BLOCK

DATA_BLOCK "RecibirVectorA"   // DB12
{ S7_Optimized_Access := 'TRUE' }
AUTHOR : SIMATIC
FAMILY : MC7Plus
NAME : TC_IP_v4
VERSION : 1.0
// stored: InstanceOfName TCON_IP_v4
"TCON_IP_v4"
BEGIN
   ID := 5;
   InterfaceId := 64;
   LocalPort := 2040;
   RemoteAddress.ADDR[1] := 192;
   RemoteAddress.ADDR[2] := 168;
   RemoteAddress.ADDR[3] := 50;
   RemoteAddress.ADDR[4] := 1;
END_DATA_BLOCK

DATA_BLOCK "EnviarVectorB"   // DB13
{ S7_Optimized_Access := 'TRUE' }
AUTHOR : SIMATIC
FAMILY : MC7Plus
NAME : TC_IP_v4
VERSION : 1.0
// stored: InstanceOfName TCON_IP_v4
"TCON_IP_v4"
BEGIN
   ID := 6;
   InterfaceId := 64;
   RemotePort := 2050;
   ActiveEstablished := true;
   RemoteAddress.ADDR[1] := 192;
   RemoteAddress.ADDR[2] := 168;
   RemoteAddress.ADDR[3] := 50;
   RemoteAddress.ADDR[4] := 1;
END_DATA_BLOCK

// folder: (top level)

ORGANIZATION_BLOCK "Main"   // OB1, LAD, ProgramCycle
TITLE = "Main Program Sweep (Cycle)"
{ S7_Optimized_Access := 'TRUE' }
VERSION : 0.1
   VAR_INPUT
      Initial_Call : Bool;   // Initial call of this OB
      Remanence : Bool;   // =True, if remanent data are available
   END_VAR
   VAR_TEMP
      col : Int;
      filas : Int;
   END_VAR
BEGIN

REGION Network 1: Enviar y Recibir modo de juego Conexion 1 y 2
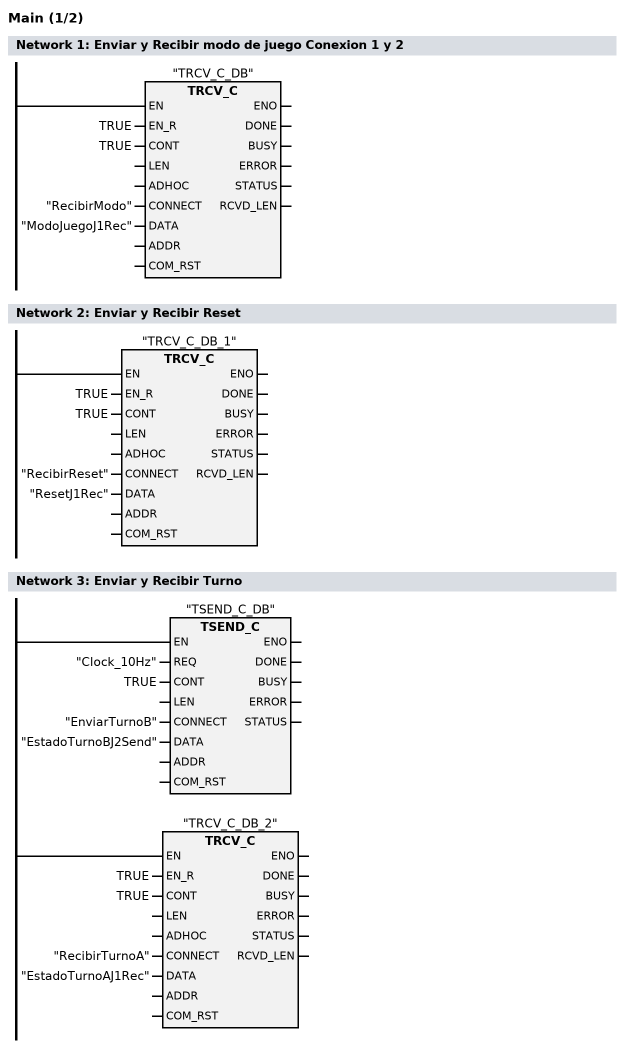
   "TRCV_C_DB"(EN_R := TRUE, CONT := TRUE, CONNECT := "RecibirModo", DATA := "ModoJuegoJ1Rec");   // TRCV_C
END_REGION

REGION Network 2: Enviar y Recibir Reset
   "TRCV_C_DB_1"(EN_R := TRUE, CONT := TRUE, CONNECT := "RecibirReset", DATA := "ResetJ1Rec");   // TRCV_C
END_REGION

REGION Network 3: Enviar y Recibir Turno
   "TSEND_C_DB"(REQ := "Clock_10Hz", CONT := TRUE, CONNECT := "EnviarTurnoB", DATA := "EstadoTurnoBJ2Send");   // TSEND_C
   "TRCV_C_DB_2"(EN_R := TRUE, CONT := TRUE, CONNECT := "RecibirTurnoA", DATA := "EstadoTurnoAJ1Rec");   // TRCV_C
END_REGION

REGION Network 4: Enviar y Recibir Turno
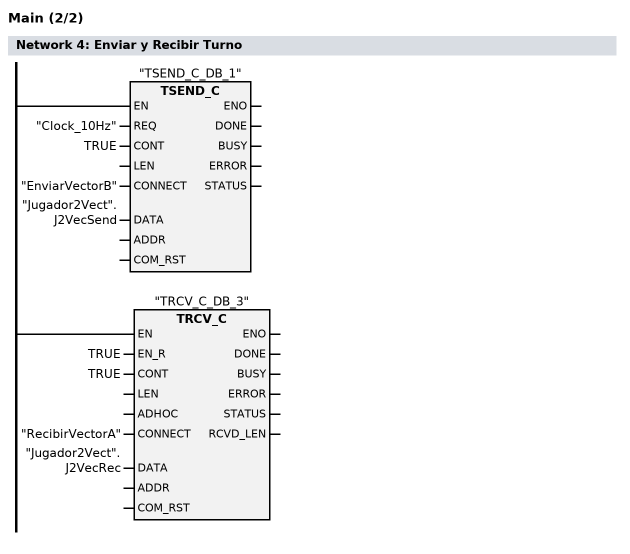
   "TSEND_C_DB_1"(REQ := "Clock_10Hz",   // TSEND_C
                  CONT := TRUE,
                  CONNECT := "EnviarVectorB",
                  DATA := "Jugador2Vect".J2VecSend);
   "TRCV_C_DB_3"(EN_R := TRUE, CONT := TRUE, CONNECT := "RecibirVectorA", DATA := "Jugador2Vect".J2VecRec);   // TRCV_C
END_REGION

REGION Network 5 (SCL): Checar si ganador rojo
   IF "ResetJ1Rec" = TRUE THEN
       "ReiniciarJ2" := TRUE;
   ELSE
       "ReiniciarJ2" := FALSE;
   END_IF;

   IF "ReiniciarJ2" = TRUE THEN
       "ModoJuegoJ2Send" := 0;
       "ModoJuegoJ1Rec" := 0;
       FILL_BLK(IN := 0,
                COUNT := 72,
                OUT => "Jugador2Vect".J2Vect[0, 0]);
       FILL_BLK(IN := 0,
                COUNT := 72,
                OUT => "Jugador2Vect".J2VecSend[0, 0]);
       FILL_BLK(IN := 0,
                COUNT := 72,
                OUT => "Jugador2Vect".J2VecRec[0, 0]);
       "Mensaje1J2" := FALSE;
       "Mensaje2J2" := FALSE;
       "Mensaje3J2" := FALSE;
       "Mensaje4J2" := FALSE;
       "Mensaje5J2" := FALSE;
       "Mensaje6J2" := FALSE;
       "Mensaje7J2" := FALSE;
       "EstadoTurnoAJ2Send" := FALSE;
       "EstadoTurnoAJ1Rec" := FALSE;
       "EstadoTurnoBJ1Rec" := FALSE;
       "EstadoTurnoBJ2Send" := FALSE;
       "Conecta4SJ2" := FALSE;
       "Conecta5SJ2" := FALSE;
       "PanelJ2" := FALSE;
       "CambioBJ2" := FALSE;
       "CambioVectorJ2" := FALSE;
   END_IF;

   IF "ModoJuegoJ1Rec" = 4 THEN
       "Conecta4SJ2" := TRUE;
       "Mensaje1J2" := TRUE;
       "Mensaje2J2" := TRUE;
       "Mensaje3J2" := FALSE;
   END_IF;

   IF "ModoJuegoJ1Rec" = 5 THEN
       "Conecta5SJ2" := TRUE;
       "Mensaje1J2" := TRUE;
       "Mensaje3J2" := TRUE;
       "Mensaje2J2" := FALSE;
   END_IF;

   IF "Conecta4SJ2" = TRUE OR "Conecta5SJ2" = TRUE THEN
       IF "EstadoTurnoAJ2Send" = TRUE THEN
           "PanelJ2" := TRUE;
           "Mensaje4J2" := TRUE;
           "Mensaje5J2" := FALSE;
       ELSE
           "PanelJ2" := FALSE;
           "Mensaje4J2" := FALSE;
           "Mensaje5J2" := TRUE;
           "CambioBJ2" := FALSE;
       END_IF;
   END_IF;

   IF "B1J2" OR "B2J2" OR "B3J2" OR "B4J2" OR "B5J2" OR "B6J2" OR "B7J2" OR "B7J2" OR "B8J2" OR "B9J2" THEN
       "EstadoTurnoBJ2Send" := TRUE;
   ELSE
       "EstadoTurnoBJ2Send" := FALSE;
   END_IF;

   IF "EstadoTurnoAJ1Rec" = TRUE THEN
       "EstadoTurnoAJ2Send" := FALSE;
   ELSIF "EstadoTurnoAJ1Rec" = FALSE THEN
       "EstadoTurnoAJ2Send" := TRUE;
   END_IF;

   IF "B1J2" AND "CambioBJ2" = FALSE THEN
       MOVE_BLK(IN := "Jugador2Vect".J2VecRec[0, 0],
                COUNT := 72,
                OUT => "Jugador2Vect".J2Vect[0, 0]);
       IF "Jugador2Vect".J2Vect[0, 0] = 0 THEN
           "Jugador2Vect".J2Vect[0, 0] := 3;
           "CambioBJ2" := TRUE;
           MOVE_BLK(IN := "Jugador2Vect".J2Vect[0, 0],
                    COUNT := 72,
                    OUT => "Jugador2Vect".J2VecSend[0, 0]);
       ELSIF "Jugador2Vect".J2Vect[1, 0] = 0 THEN
           "Jugador2Vect".J2Vect[1, 0] := 3;
           "CambioBJ2" := TRUE;
           MOVE_BLK(IN := "Jugador2Vect".J2Vect[0, 0],
                    COUNT := 72,
                    OUT => "Jugador2Vect".J2VecSend[0, 0]);
       ELSIF "Jugador2Vect".J2Vect[2, 0] = 0 THEN
           "Jugador2Vect".J2Vect[2, 0] := 3;
           "CambioBJ2" := TRUE;
           MOVE_BLK(IN := "Jugador2Vect".J2Vect[0, 0],
                    COUNT := 72,
                    OUT => "Jugador2Vect".J2VecSend[0, 0]);
       ELSIF "Jugador2Vect".J2Vect[3, 0] = 0 THEN
           "Jugador2Vect".J2Vect[3, 0] := 3;
           "CambioBJ2" := TRUE;
           MOVE_BLK(IN := "Jugador2Vect".J2Vect[0, 0],
                    COUNT := 72,
                    OUT => "Jugador2Vect".J2VecSend[0, 0]);
       ELSIF "Jugador2Vect".J2Vect[4, 0] = 0 THEN
           "Jugador2Vect".J2Vect[4, 0] := 3;
           "CambioBJ2" := TRUE;
           MOVE_BLK(IN := "Jugador2Vect".J2Vect[0, 0],
                    COUNT := 72,
                    OUT => "Jugador2Vect".J2VecSend[0, 0]);
       ELSIF "Jugador2Vect".J2Vect[5, 0] = 0 THEN
           "Jugador2Vect".J2Vect[5, 0] := 3;
           "CambioBJ2" := TRUE;
           MOVE_BLK(IN := "Jugador2Vect".J2Vect[0, 0],
                    COUNT := 72,
                    OUT => "Jugador2Vect".J2VecSend[0, 0]);
       ELSIF "Jugador2Vect".J2Vect[6, 0] = 0 THEN
           "Jugador2Vect".J2Vect[6, 0] := 3;
           "CambioBJ2" := TRUE;
           MOVE_BLK(IN := "Jugador2Vect".J2Vect[0, 0],
                    COUNT := 72,
                    OUT => "Jugador2Vect".J2VecSend[0, 0]);
       ELSIF "Jugador2Vect".J2Vect[7, 0] = 0 THEN
           "Jugador2Vect".J2Vect[7, 0] := 3;
           "CambioBJ2" := TRUE;
           MOVE_BLK(IN := "Jugador2Vect".J2Vect[0, 0],
                    COUNT := 72,
                    OUT => "Jugador2Vect".J2VecSend[0, 0]);
       END_IF;
   END_IF;


   IF "B2J2" AND "CambioBJ2" = FALSE THEN
       MOVE_BLK(IN := "Jugador2Vect".J2VecRec[0, 0],
                COUNT := 72,
                OUT => "Jugador2Vect".J2Vect[0, 0]);
       IF "Jugador2Vect".J2Vect[0, 1] = 0 THEN
           "Jugador2Vect".J2Vect[0, 1] := 3;
           "CambioBJ2" := TRUE;
           MOVE_BLK(IN := "Jugador2Vect".J2Vect[0, 0],
                    COUNT := 72,
                    OUT => "Jugador2Vect".J2VecSend[0, 0]);
       ELSIF "Jugador2Vect".J2Vect[1, 1] = 0 THEN
           "Jugador2Vect".J2Vect[1, 1] := 3;
           "CambioBJ2" := TRUE;
           MOVE_BLK(IN := "Jugador2Vect".J2Vect[0, 0],
                    COUNT := 72,
                    OUT => "Jugador2Vect".J2VecSend[0, 0]);
       ELSIF "Jugador2Vect".J2Vect[2, 1] = 0 THEN
           "Jugador2Vect".J2Vect[2, 1] := 3;
           "CambioBJ2" := TRUE;
           MOVE_BLK(IN := "Jugador2Vect".J2Vect[0, 0],
                    COUNT := 72,
                    OUT => "Jugador2Vect".J2VecSend[0, 0]);
       ELSIF "Jugador2Vect".J2Vect[3, 1] = 0 THEN
           "Jugador2Vect".J2Vect[3, 1] := 3;
           "CambioBJ2" := TRUE;
           MOVE_BLK(IN := "Jugador2Vect".J2Vect[0, 0],
                    COUNT := 72,
                    OUT => "Jugador2Vect".J2VecSend[0, 0]);
       ELSIF "Jugador2Vect".J2Vect[4, 1] = 0 THEN
           "Jugador2Vect".J2Vect[4, 1] := 3;
           "CambioBJ2" := TRUE;
           MOVE_BLK(IN := "Jugador2Vect".J2Vect[0, 0],
                    COUNT := 72,
                    OUT => "Jugador2Vect".J2VecSend[0, 0]);
       ELSIF "Jugador2Vect".J2Vect[5, 1] = 0 THEN
           "Jugador2Vect".J2Vect[5, 1] := 3;
           "CambioBJ2" := TRUE;
           MOVE_BLK(IN := "Jugador2Vect".J2Vect[0, 0],
                    COUNT := 72,
                    OUT => "Jugador2Vect".J2VecSend[0, 0]);
       ELSIF "Jugador2Vect".J2Vect[6, 1] = 0 THEN
           "Jugador2Vect".J2Vect[6, 1] := 3;
           "CambioBJ2" := TRUE;
           MOVE_BLK(IN := "Jugador2Vect".J2Vect[0, 0],
                    COUNT := 72,
                    OUT => "Jugador2Vect".J2VecSend[0, 0]);
       ELSIF "Jugador2Vect".J2Vect[7, 1] = 0 THEN
           "Jugador2Vect".J2Vect[7, 1] := 3;
           "CambioBJ2" := TRUE;
           MOVE_BLK(IN := "Jugador2Vect".J2Vect[0, 0],
                    COUNT := 72,
                    OUT => "Jugador2Vect".J2VecSend[0, 0]);
       END_IF;
   END_IF;


   IF "B3J2" AND "CambioBJ2" = FALSE THEN
       MOVE_BLK(IN := "Jugador2Vect".J2VecRec[0, 0],
                COUNT := 72,
                OUT => "Jugador2Vect".J2Vect[0, 0]);
       IF "Jugador2Vect".J2Vect[0, 2] = 0 THEN
           "Jugador2Vect".J2Vect[0, 2] := 3;
           "CambioBJ2" := TRUE;
           MOVE_BLK(IN := "Jugador2Vect".J2Vect[0, 0],
                    COUNT := 72,
                    OUT => "Jugador2Vect".J2VecSend[0, 0]);
       ELSIF "Jugador2Vect".J2Vect[1, 2] = 0 THEN
           "Jugador2Vect".J2Vect[1, 2] := 3;
           "CambioBJ2" := TRUE;
           MOVE_BLK(IN := "Jugador2Vect".J2Vect[0, 0],
                    COUNT := 72,
                    OUT => "Jugador2Vect".J2VecSend[0, 0]);
       ELSIF "Jugador2Vect".J2Vect[2, 2] = 0 THEN
           "Jugador2Vect".J2Vect[2, 2] := 3;
           "CambioBJ2" := TRUE;
           MOVE_BLK(IN := "Jugador2Vect".J2Vect[0, 0],
                    COUNT := 72,
                    OUT => "Jugador2Vect".J2VecSend[0, 0]);
       ELSIF "Jugador2Vect".J2Vect[3, 2] = 0 THEN
           "Jugador2Vect".J2Vect[3, 2] := 3;
           "CambioBJ2" := TRUE;
           MOVE_BLK(IN := "Jugador2Vect".J2Vect[0, 0],
                    COUNT := 72,
                    OUT => "Jugador2Vect".J2VecSend[0, 0]);
       ELSIF "Jugador2Vect".J2Vect[4, 2] = 0 THEN
           "Jugador2Vect".J2Vect[4, 2] := 3;
           "CambioBJ2" := TRUE;
           MOVE_BLK(IN := "Jugador2Vect".J2Vect[0, 0],
                    COUNT := 72,
                    OUT => "Jugador2Vect".J2VecSend[0, 0]);
       ELSIF "Jugador2Vect".J2Vect[5, 2] = 0 THEN
           "Jugador2Vect".J2Vect[5, 2] := 3;
           "CambioBJ2" := TRUE;
           MOVE_BLK(IN := "Jugador2Vect".J2Vect[0, 0],
                    COUNT := 72,
                    OUT => "Jugador2Vect".J2VecSend[0, 0]);
       ELSIF "Jugador2Vect".J2Vect[6, 2] = 0 THEN
           "Jugador2Vect".J2Vect[6, 2] := 3;
           "CambioBJ2" := TRUE;
           MOVE_BLK(IN := "Jugador2Vect".J2Vect[0, 0],
                    COUNT := 72,
                    OUT => "Jugador2Vect".J2VecSend[0, 0]);
       ELSIF "Jugador2Vect".J2Vect[7, 2] = 0 THEN
           "Jugador2Vect".J2Vect[7, 2] := 3;
           "CambioBJ2" := TRUE;
           MOVE_BLK(IN := "Jugador2Vect".J2Vect[0, 0],
                    COUNT := 72,
                    OUT => "Jugador2Vect".J2VecSend[0, 0]);
       END_IF;
   END_IF;


   IF "B4J2" AND "CambioBJ2" = FALSE THEN
       MOVE_BLK(IN := "Jugador2Vect".J2VecRec[0, 0],
                COUNT := 72,
                OUT => "Jugador2Vect".J2Vect[0, 0]);
       IF "Jugador2Vect".J2Vect[0, 3] = 0 THEN
           "Jugador2Vect".J2Vect[0, 3] := 3;
           "CambioBJ2" := TRUE;
           MOVE_BLK(IN := "Jugador2Vect".J2Vect[0, 0],
                    COUNT := 72,
                    OUT => "Jugador2Vect".J2VecSend[0, 0]);
       ELSIF "Jugador2Vect".J2Vect[1, 3] = 0 THEN
           "Jugador2Vect".J2Vect[1, 3] := 3;
           "CambioBJ2" := TRUE;
           MOVE_BLK(IN := "Jugador2Vect".J2Vect[0, 0],
                    COUNT := 72,
                    OUT => "Jugador2Vect".J2VecSend[0, 0]);
       ELSIF "Jugador2Vect".J2Vect[2, 3] = 0 THEN
           "Jugador2Vect".J2Vect[2, 3] := 3;
           "CambioBJ2" := TRUE;
           MOVE_BLK(IN := "Jugador2Vect".J2Vect[0, 0],
                    COUNT := 72,
                    OUT => "Jugador2Vect".J2VecSend[0, 0]);
       ELSIF "Jugador2Vect".J2Vect[3, 3] = 0 THEN
           "Jugador2Vect".J2Vect[3, 3] := 3;
           "CambioBJ2" := TRUE;
           MOVE_BLK(IN := "Jugador2Vect".J2Vect[0, 0],
                    COUNT := 72,
                    OUT => "Jugador2Vect".J2VecSend[0, 0]);
       ELSIF "Jugador2Vect".J2Vect[4, 3] = 0 THEN
           "Jugador2Vect".J2Vect[4, 3] := 3;
           "CambioBJ2" := TRUE;
           MOVE_BLK(IN := "Jugador2Vect".J2Vect[0, 0],
                    COUNT := 72,
                    OUT => "Jugador2Vect".J2VecSend[0, 0]);
       ELSIF "Jugador2Vect".J2Vect[5, 3] = 0 THEN
           "Jugador2Vect".J2Vect[5, 3] := 3;
           "CambioBJ2" := TRUE;
           MOVE_BLK(IN := "Jugador2Vect".J2Vect[0, 0],
                    COUNT := 72,
                    OUT => "Jugador2Vect".J2VecSend[0, 0]);
       ELSIF "Jugador2Vect".J2Vect[6, 3] = 0 THEN
           "Jugador2Vect".J2Vect[6, 3] := 3;
           "CambioBJ2" := TRUE;
           MOVE_BLK(IN := "Jugador2Vect".J2Vect[0, 0],
                    COUNT := 72,
                    OUT => "Jugador2Vect".J2VecSend[0, 0]);
       ELSIF "Jugador2Vect".J2Vect[7, 3] = 0 THEN
           "Jugador2Vect".J2Vect[7, 3] := 3;
           "CambioBJ2" := TRUE;
           MOVE_BLK(IN := "Jugador2Vect".J2Vect[0, 0],
                    COUNT := 72,
                    OUT => "Jugador2Vect".J2VecSend[0, 0]);
       END_IF;
   END_IF;


   IF "B5J2" AND "CambioBJ2" = FALSE THEN
       MOVE_BLK(IN := "Jugador2Vect".J2VecRec[0, 0],
                COUNT := 72,
                OUT => "Jugador2Vect".J2Vect[0, 0]);
       IF "Jugador2Vect".J2Vect[0, 4] = 0 THEN
           "Jugador2Vect".J2Vect[0, 4] := 3;
           "CambioBJ2" := TRUE;
           MOVE_BLK(IN := "Jugador2Vect".J2Vect[0, 0],
                    COUNT := 72,
                    OUT => "Jugador2Vect".J2VecSend[0, 0]);
       ELSIF "Jugador2Vect".J2Vect[1, 4] = 0 THEN
           "Jugador2Vect".J2Vect[1, 4] := 3;
           "CambioBJ2" := TRUE;
           MOVE_BLK(IN := "Jugador2Vect".J2Vect[0, 0],
                    COUNT := 72,
                    OUT => "Jugador2Vect".J2VecSend[0, 0]);
       ELSIF "Jugador2Vect".J2Vect[2, 4] = 0 THEN
           "Jugador2Vect".J2Vect[2, 4] := 3;
           "CambioBJ2" := TRUE;
           MOVE_BLK(IN := "Jugador2Vect".J2Vect[0, 0],
                    COUNT := 72,
                    OUT => "Jugador2Vect".J2VecSend[0, 0]);
       ELSIF "Jugador2Vect".J2Vect[3, 4] = 0 THEN
           "Jugador2Vect".J2Vect[3, 4] := 3;
           "CambioBJ2" := TRUE;
           MOVE_BLK(IN := "Jugador2Vect".J2Vect[0, 0],
                    COUNT := 72,
                    OUT => "Jugador2Vect".J2VecSend[0, 0]);
       ELSIF "Jugador2Vect".J2Vect[4, 4] = 0 THEN
           "Jugador2Vect".J2Vect[4, 4] := 3;
           "CambioBJ2" := TRUE;
           MOVE_BLK(IN := "Jugador2Vect".J2Vect[0, 0],
                    COUNT := 72,
                    OUT => "Jugador2Vect".J2VecSend[0, 0]);
       ELSIF "Jugador2Vect".J2Vect[5, 4] = 0 THEN
           "Jugador2Vect".J2Vect[5, 4] := 3;
           "CambioBJ2" := TRUE;
           MOVE_BLK(IN := "Jugador2Vect".J2Vect[0, 0],
                    COUNT := 72,
                    OUT => "Jugador2Vect".J2VecSend[0, 0]);
       ELSIF "Jugador2Vect".J2Vect[6, 4] = 0 THEN
           "Jugador2Vect".J2Vect[6, 4] := 3;
           "CambioBJ2" := TRUE;
           MOVE_BLK(IN := "Jugador2Vect".J2Vect[0, 0],
                    COUNT := 72,
                    OUT => "Jugador2Vect".J2VecSend[0, 0]);
       ELSIF "Jugador2Vect".J2Vect[7, 4] = 0 THEN
           "Jugador2Vect".J2Vect[7, 4] := 3;
           "CambioBJ2" := TRUE;
           MOVE_BLK(IN := "Jugador2Vect".J2Vect[0, 0],
                    COUNT := 72,
                    OUT => "Jugador2Vect".J2VecSend[0, 0]);
       END_IF;
   END_IF;


   IF "B6J2" AND "CambioBJ2" = FALSE THEN
       MOVE_BLK(IN := "Jugador2Vect".J2VecRec[0, 0],
                COUNT := 72,
                OUT => "Jugador2Vect".J2Vect[0, 0]);
       IF "Jugador2Vect".J2Vect[0, 5] = 0 THEN
           "Jugador2Vect".J2Vect[0, 5] := 3;
           "CambioBJ2" := TRUE;
           MOVE_BLK(IN := "Jugador2Vect".J2Vect[0, 0],
                    COUNT := 72,
                    OUT => "Jugador2Vect".J2VecSend[0, 0]);
       ELSIF "Jugador2Vect".J2Vect[1, 5] = 0 THEN
           "Jugador2Vect".J2Vect[1, 5] := 3;
           "CambioBJ2" := TRUE;
           MOVE_BLK(IN := "Jugador2Vect".J2Vect[0, 0],
                    COUNT := 72,
                    OUT => "Jugador2Vect".J2VecSend[0, 0]);
       ELSIF "Jugador2Vect".J2Vect[2, 5] = 0 THEN
           "Jugador2Vect".J2Vect[2, 5] := 3;
           "CambioBJ2" := TRUE;
           MOVE_BLK(IN := "Jugador2Vect".J2Vect[0, 0],
                    COUNT := 72,
                    OUT => "Jugador2Vect".J2VecSend[0, 0]);
       ELSIF "Jugador2Vect".J2Vect[3, 5] = 0 THEN
           "Jugador2Vect".J2Vect[3, 5] := 3;
           "CambioBJ2" := TRUE;
           MOVE_BLK(IN := "Jugador2Vect".J2Vect[0, 0],
                    COUNT := 72,
                    OUT => "Jugador2Vect".J2VecSend[0, 0]);
       ELSIF "Jugador2Vect".J2Vect[4, 5] = 0 THEN
           "Jugador2Vect".J2Vect[4, 5] := 3;
           "CambioBJ2" := TRUE;
           MOVE_BLK(IN := "Jugador2Vect".J2Vect[0, 0],
                    COUNT := 72,
                    OUT => "Jugador2Vect".J2VecSend[0, 0]);
       ELSIF "Jugador2Vect".J2Vect[5, 5] = 0 THEN
           "Jugador2Vect".J2Vect[5, 5] := 3;
           "CambioBJ2" := TRUE;
           MOVE_BLK(IN := "Jugador2Vect".J2Vect[0, 0],
                    COUNT := 72,
                    OUT => "Jugador2Vect".J2VecSend[0, 0]);
       ELSIF "Jugador2Vect".J2Vect[6, 5] = 0 THEN
           "Jugador2Vect".J2Vect[6, 5] := 3;
           "CambioBJ2" := TRUE;
           MOVE_BLK(IN := "Jugador2Vect".J2Vect[0, 0],
                    COUNT := 72,
                    OUT => "Jugador2Vect".J2VecSend[0, 0]);
       ELSIF "Jugador2Vect".J2Vect[7, 5] = 0 THEN
           "Jugador2Vect".J2Vect[7, 5] := 3;
           "CambioBJ2" := TRUE;
           MOVE_BLK(IN := "Jugador2Vect".J2Vect[0, 0],
                    COUNT := 72,
                    OUT => "Jugador2Vect".J2VecSend[0, 0]);
       END_IF;
   END_IF;


   IF "B7J2" AND "CambioBJ2" = FALSE THEN
       MOVE_BLK(IN := "Jugador2Vect".J2VecRec[0, 0],
                COUNT := 72,
                OUT => "Jugador2Vect".J2Vect[0, 0]);
       IF "Jugador2Vect".J2Vect[0, 6] = 0 THEN
           "Jugador2Vect".J2Vect[0, 6] := 3;
           "CambioBJ2" := TRUE;
           MOVE_BLK(IN := "Jugador2Vect".J2Vect[0, 0],
                    COUNT := 72,
                    OUT => "Jugador2Vect".J2VecSend[0, 0]);
       ELSIF "Jugador2Vect".J2Vect[1, 6] = 0 THEN
           "Jugador2Vect".J2Vect[1, 6] := 3;
           "CambioBJ2" := TRUE;
           MOVE_BLK(IN := "Jugador2Vect".J2Vect[0, 0],
                    COUNT := 72,
                    OUT => "Jugador2Vect".J2VecSend[0, 0]);
       ELSIF "Jugador2Vect".J2Vect[2, 6] = 0 THEN
           "Jugador2Vect".J2Vect[2, 6] := 3;
           "CambioBJ2" := TRUE;
           MOVE_BLK(IN := "Jugador2Vect".J2Vect[0, 0],
                    COUNT := 72,
                    OUT => "Jugador2Vect".J2VecSend[0, 0]);
       ELSIF "Jugador2Vect".J2Vect[3, 6] = 0 THEN
           "Jugador2Vect".J2Vect[3, 6] := 3;
           "CambioBJ2" := TRUE;
           MOVE_BLK(IN := "Jugador2Vect".J2Vect[0, 0],
                    COUNT := 72,
                    OUT => "Jugador2Vect".J2VecSend[0, 0]);
       ELSIF "Jugador2Vect".J2Vect[4, 6] = 0 THEN
           "Jugador2Vect".J2Vect[4, 6] := 3;
           "CambioBJ2" := TRUE;
           MOVE_BLK(IN := "Jugador2Vect".J2Vect[0, 0],
                    COUNT := 72,
                    OUT => "Jugador2Vect".J2VecSend[0, 0]);
       ELSIF "Jugador2Vect".J2Vect[5, 6] = 0 THEN
           "Jugador2Vect".J2Vect[5, 6] := 3;
           "CambioBJ2" := TRUE;
           MOVE_BLK(IN := "Jugador2Vect".J2Vect[0, 0],
                    COUNT := 72,
                    OUT => "Jugador2Vect".J2VecSend[0, 0]);
       ELSIF "Jugador2Vect".J2Vect[6, 6] = 0 THEN
           "Jugador2Vect".J2Vect[6, 6] := 3;
           "CambioBJ2" := TRUE;
           MOVE_BLK(IN := "Jugador2Vect".J2Vect[0, 0],
                    COUNT := 72,
                    OUT => "Jugador2Vect".J2VecSend[0, 0]);
       ELSIF "Jugador2Vect".J2Vect[7, 6] = 0 THEN
           "Jugador2Vect".J2Vect[7, 6] := 3;
           "CambioBJ2" := TRUE;
           MOVE_BLK(IN := "Jugador2Vect".J2Vect[0, 0],
                    COUNT := 72,
                    OUT => "Jugador2Vect".J2VecSend[0, 0]);
       END_IF;
   END_IF;


   IF "B8J2" AND "CambioBJ2" = FALSE THEN
       MOVE_BLK(IN := "Jugador2Vect".J2VecRec[0, 0],
                COUNT := 72,
                OUT => "Jugador2Vect".J2Vect[0, 0]);
       IF "Jugador2Vect".J2Vect[0, 7] = 0 THEN
           "Jugador2Vect".J2Vect[0, 7] := 3;
           "CambioBJ2" := TRUE;
           MOVE_BLK(IN := "Jugador2Vect".J2Vect[0, 0],
                    COUNT := 72,
                    OUT => "Jugador2Vect".J2VecSend[0, 0]);
       ELSIF "Jugador2Vect".J2Vect[1, 7] = 0 THEN
           "Jugador2Vect".J2Vect[1, 7] := 3;
           "CambioBJ2" := TRUE;
           MOVE_BLK(IN := "Jugador2Vect".J2Vect[0, 0],
                    COUNT := 72,
                    OUT => "Jugador2Vect".J2VecSend[0, 0]);
       ELSIF "Jugador2Vect".J2Vect[2, 7] = 0 THEN
           "Jugador2Vect".J2Vect[2, 7] := 3;
           "CambioBJ2" := TRUE;
           MOVE_BLK(IN := "Jugador2Vect".J2Vect[0, 0],
                    COUNT := 72,
                    OUT => "Jugador2Vect".J2VecSend[0, 0]);
       ELSIF "Jugador2Vect".J2Vect[3, 7] = 0 THEN
           "Jugador2Vect".J2Vect[3, 7] := 3;
           "CambioBJ2" := TRUE;
           MOVE_BLK(IN := "Jugador2Vect".J2Vect[0, 0],
                    COUNT := 72,
                    OUT => "Jugador2Vect".J2VecSend[0, 0]);
       ELSIF "Jugador2Vect".J2Vect[4, 7] = 0 THEN
           "Jugador2Vect".J2Vect[4, 7] := 3;
           "CambioBJ2" := TRUE;
           MOVE_BLK(IN := "Jugador2Vect".J2Vect[0, 0],
                    COUNT := 72,
                    OUT => "Jugador2Vect".J2VecSend[0, 0]);
       ELSIF "Jugador2Vect".J2Vect[5, 7] = 0 THEN
           "Jugador2Vect".J2Vect[5, 7] := 3;
           "CambioBJ2" := TRUE;
           MOVE_BLK(IN := "Jugador2Vect".J2Vect[0, 0],
                    COUNT := 72,
                    OUT => "Jugador2Vect".J2VecSend[0, 0]);
       ELSIF "Jugador2Vect".J2Vect[6, 7] = 0 THEN
           "Jugador2Vect".J2Vect[6, 7] := 3;
           "CambioBJ2" := TRUE;
           MOVE_BLK(IN := "Jugador2Vect".J2Vect[0, 0],
                    COUNT := 72,
                    OUT => "Jugador2Vect".J2VecSend[0, 0]);
       ELSIF "Jugador2Vect".J2Vect[7, 7] = 0 THEN
           "Jugador2Vect".J2Vect[7, 7] := 3;
           "CambioBJ2" := TRUE;
           MOVE_BLK(IN := "Jugador2Vect".J2Vect[0, 0],
                    COUNT := 72,
                    OUT => "Jugador2Vect".J2VecSend[0, 0]);
       END_IF;
   END_IF;


   IF "B9J2" AND "CambioBJ2" = FALSE THEN
       MOVE_BLK(IN := "Jugador2Vect".J2VecRec[0, 0],
                COUNT := 72,
                OUT => "Jugador2Vect".J2Vect[0, 0]);
       IF "Jugador2Vect".J2Vect[0, 8] = 0 THEN
           "Jugador2Vect".J2Vect[0, 8] := 3;
           "CambioBJ2" := TRUE;
           MOVE_BLK(IN := "Jugador2Vect".J2Vect[0, 0],
                    COUNT := 72,
                    OUT => "Jugador2Vect".J2VecSend[0, 0]);
       ELSIF "Jugador2Vect".J2Vect[1, 8] = 0 THEN
           "Jugador2Vect".J2Vect[1, 8] := 3;
           "CambioBJ2" := TRUE;
           MOVE_BLK(IN := "Jugador2Vect".J2Vect[0, 0],
                    COUNT := 72,
                    OUT => "Jugador2Vect".J2VecSend[0, 0]);
       ELSIF "Jugador2Vect".J2Vect[2, 8] = 0 THEN
           "Jugador2Vect".J2Vect[2, 8] := 3;
           "CambioBJ2" := TRUE;
           MOVE_BLK(IN := "Jugador2Vect".J2Vect[0, 0],
                    COUNT := 72,
                    OUT => "Jugador2Vect".J2VecSend[0, 0]);
       ELSIF "Jugador2Vect".J2Vect[3, 8] = 0 THEN
           "Jugador2Vect".J2Vect[3, 8] := 3;
           "CambioBJ2" := TRUE;
           MOVE_BLK(IN := "Jugador2Vect".J2Vect[0, 0],
                    COUNT := 72,
                    OUT => "Jugador2Vect".J2VecSend[0, 0]);
       ELSIF "Jugador2Vect".J2Vect[4, 8] = 0 THEN
           "Jugador2Vect".J2Vect[4, 8] := 3;
           "CambioBJ2" := TRUE;
           MOVE_BLK(IN := "Jugador2Vect".J2Vect[0, 0],
                    COUNT := 72,
                    OUT => "Jugador2Vect".J2VecSend[0, 0]);
       ELSIF "Jugador2Vect".J2Vect[5, 8] = 0 THEN
           "Jugador2Vect".J2Vect[5, 8] := 3;
           "CambioBJ2" := TRUE;
           MOVE_BLK(IN := "Jugador2Vect".J2Vect[0, 0],
                    COUNT := 72,
                    OUT => "Jugador2Vect".J2VecSend[0, 0]);
       ELSIF "Jugador2Vect".J2Vect[6, 8] = 0 THEN
           "Jugador2Vect".J2Vect[6, 8] := 3;
           "CambioBJ2" := TRUE;
           MOVE_BLK(IN := "Jugador2Vect".J2Vect[0, 0],
                    COUNT := 72,
                    OUT => "Jugador2Vect".J2VecSend[0, 0]);
       ELSIF "Jugador2Vect".J2Vect[7, 8] = 0 THEN
           "Jugador2Vect".J2Vect[7, 8] := 3;
           "CambioBJ2" := TRUE;
           MOVE_BLK(IN := "Jugador2Vect".J2Vect[0, 0],
                    COUNT := 72,
                    OUT => "Jugador2Vect".J2VecSend[0, 0]);
       END_IF;
   END_IF;


   IF ("B1J2" = FALSE OR "B2J2" = FALSE OR "B3J2" = FALSE OR "B4J2" = FALSE OR "B5J2" = FALSE OR "B6J2" = FALSE OR "B7J2" = FALSE OR "B8J2" = FALSE OR "B9J2" = FALSE) AND "CambioBJ2" = TRUE THEN
       "CambioBJ2" := FALSE;
       "CambioVectorJ2" := FALSE;
   END_IF;
END_REGION
END_ORGANIZATION_BLOCK

(* ===== HMI "HMI_RT_1" =====
system functions are stored by id; their names below are inferred from use
connection "HMI_Connection_1": ETHERNET, S7_1500_OMS

HMI tags "Default tag table"
   "Tag_ScreenNumber" : UInt, internal
   "Mensaje1J1" : Bool = PLC Mensaje1J1 AT %M11.0, 1 s
   "Mensaje2J1" : Bool = PLC Mensaje2J1 AT %M11.1, 1 s
   "Mensaje3J1" : Bool = PLC Mensaje3J1 AT %M11.2, 1 s
   "Mensaje4J1" : Bool = PLC Mensaje4J1 AT %M11.3, 1 s
   "Mensaje5J1" : Bool = PLC Mensaje5J1 AT %M11.4, 1 s
   "Mensaje6J1" : Bool = PLC Mensaje6J1 AT %M11.5, 1 s
   "Mensaje7J1" : Bool = PLC Mensaje7J1 AT %M11.6, 1 s
   "PanelJ1" : Bool = PLC PanelJ1 AT %M13.0, 1 s
   "B1J1" : Bool = PLC B1J1 AT %M11.7, 1 s
   "B2J1" : Bool = PLC B2J1 AT %M12.0, 1 s
   "B3J1" : Bool = PLC B3J1 AT %M12.1, 1 s
   "B4J1" : Bool = PLC B4J1 AT %M12.2, 1 s
   "B5J1" : Bool = PLC B5J1 AT %M12.3, 1 s
   "B6J1" : Bool = PLC B6J1 AT %M12.4, 1 s
   "B7J1" : Bool = PLC B7J1 AT %M12.5, 1 s
   "B8J1" : Bool = PLC B8J1 AT %M12.6, 1 s
   "B9J1" : Bool = PLC B9J1 AT %M12.7, 1 s
   "Jugador1Vect_J1Vect{0,0}" : Int = PLC Jugador1Vect.J1Vect[0,0] AT %DB4.DBW0, 1 s
   "Jugador1Vect_J1Vect{0,1}" : Int = PLC Jugador1Vect.J1Vect[0,1] AT %DB4.DBW2, 1 s
   "Jugador1Vect_J1Vect{0,2}" : Int = PLC Jugador1Vect.J1Vect[0,2] AT %DB4.DBW4, 1 s
   "Jugador1Vect_J1Vect{0,3}" : Int = PLC Jugador1Vect.J1Vect[0,3] AT %DB4.DBW6, 1 s
   "Jugador1Vect_J1Vect{0,4}" : Int = PLC Jugador1Vect.J1Vect[0,4] AT %DB4.DBW8, 1 s
   "Jugador1Vect_J1Vect{0,5}" : Int = PLC Jugador1Vect.J1Vect[0,5] AT %DB4.DBW10, 1 s
   "Jugador1Vect_J1Vect{0,6}" : Int = PLC Jugador1Vect.J1Vect[0,6] AT %DB4.DBW12, 1 s
   "Jugador1Vect_J1Vect{0,7}" : Int = PLC Jugador1Vect.J1Vect[0,7] AT %DB4.DBW14, 1 s
   "Jugador1Vect_J1Vect{0,8}" : Int = PLC Jugador1Vect.J1Vect[0,8] AT %DB4.DBW16, 1 s
   "Jugador1Vect_J1Vect{1,0}" : Int = PLC Jugador1Vect.J1Vect[1,0] AT %DB4.DBW18, 1 s
   "Jugador1Vect_J1Vect{1,1}" : Int = PLC Jugador1Vect.J1Vect[1,1] AT %DB4.DBW20, 1 s
   "Jugador1Vect_J1Vect{1,2}" : Int = PLC Jugador1Vect.J1Vect[1,2] AT %DB4.DBW22, 1 s
   "Jugador1Vect_J1Vect{1,3}" : Int = PLC Jugador1Vect.J1Vect[1,3] AT %DB4.DBW24, 1 s
   "Jugador1Vect_J1Vect{1,4}" : Int = PLC Jugador1Vect.J1Vect[1,4] AT %DB4.DBW26, 1 s
   "Jugador1Vect_J1Vect{1,5}" : Int = PLC Jugador1Vect.J1Vect[1,5] AT %DB4.DBW28, 1 s
   "Jugador1Vect_J1Vect{1,6}" : Int = PLC Jugador1Vect.J1Vect[1,6] AT %DB4.DBW30, 1 s
   "Jugador1Vect_J1Vect{1,7}" : Int = PLC Jugador1Vect.J1Vect[1,7] AT %DB4.DBW32, 1 s
   "Jugador1Vect_J1Vect{1,8}" : Int = PLC Jugador1Vect.J1Vect[1,8] AT %DB4.DBW34, 1 s
   "Jugador1Vect_J1Vect{2,0}" : Int = PLC Jugador1Vect.J1Vect[2,0] AT %DB4.DBW36, 1 s
   "Jugador1Vect_J1Vect{2,1}" : Int = PLC Jugador1Vect.J1Vect[2,1] AT %DB4.DBW38, 1 s
   "Jugador1Vect_J1Vect{2,2}" : Int = PLC Jugador1Vect.J1Vect[2,2] AT %DB4.DBW40, 1 s
   "Jugador1Vect_J1Vect{2,3}" : Int = PLC Jugador1Vect.J1Vect[2,3] AT %DB4.DBW42, 1 s
   "Jugador1Vect_J1Vect{2,4}" : Int = PLC Jugador1Vect.J1Vect[2,4] AT %DB4.DBW44, 1 s
   "Jugador1Vect_J1Vect{2,5}" : Int = PLC Jugador1Vect.J1Vect[2,5] AT %DB4.DBW46, 1 s
   "Jugador1Vect_J1Vect{2,6}" : Int = PLC Jugador1Vect.J1Vect[2,6] AT %DB4.DBW48, 1 s
   "Jugador1Vect_J1Vect{2,7}" : Int = PLC Jugador1Vect.J1Vect[2,7] AT %DB4.DBW50, 1 s
   "Jugador1Vect_J1Vect{2,8}" : Int = PLC Jugador1Vect.J1Vect[2,8] AT %DB4.DBW52, 1 s
   "Jugador1Vect_J1Vect{3,0}" : Int = PLC Jugador1Vect.J1Vect[3,0] AT %DB4.DBW54, 1 s
   "Jugador1Vect_J1Vect{3,1}" : Int = PLC Jugador1Vect.J1Vect[3,1] AT %DB4.DBW56, 1 s
   "Jugador1Vect_J1Vect{3,2}" : Int = PLC Jugador1Vect.J1Vect[3,2] AT %DB4.DBW58, 1 s
   "Jugador1Vect_J1Vect{3,3}" : Int = PLC Jugador1Vect.J1Vect[3,3] AT %DB4.DBW60, 1 s
   "Jugador1Vect_J1Vect{3,4}" : Int = PLC Jugador1Vect.J1Vect[3,4] AT %DB4.DBW62, 1 s
   "Jugador1Vect_J1Vect{3,5}" : Int = PLC Jugador1Vect.J1Vect[3,5] AT %DB4.DBW64, 1 s
   "Jugador1Vect_J1Vect{3,6}" : Int = PLC Jugador1Vect.J1Vect[3,6] AT %DB4.DBW66, 1 s
   "Jugador1Vect_J1Vect{3,7}" : Int = PLC Jugador1Vect.J1Vect[3,7] AT %DB4.DBW68, 1 s
   "Jugador1Vect_J1Vect{3,8}" : Int = PLC Jugador1Vect.J1Vect[3,8] AT %DB4.DBW70, 1 s
   "Jugador1Vect_J1Vect{4,0}" : Int = PLC Jugador1Vect.J1Vect[4,0] AT %DB4.DBW72, 1 s
   "Jugador1Vect_J1Vect{4,1}" : Int = PLC Jugador1Vect.J1Vect[4,1] AT %DB4.DBW74, 1 s
   "Jugador1Vect_J1Vect{4,2}" : Int = PLC Jugador1Vect.J1Vect[4,2] AT %DB4.DBW76, 1 s
   "Jugador1Vect_J1Vect{4,3}" : Int = PLC Jugador1Vect.J1Vect[4,3] AT %DB4.DBW78, 1 s
   "Jugador1Vect_J1Vect{4,4}" : Int = PLC Jugador1Vect.J1Vect[4,4] AT %DB4.DBW80, 1 s
   "Jugador1Vect_J1Vect{4,5}" : Int = PLC Jugador1Vect.J1Vect[4,5] AT %DB4.DBW82, 1 s
   "Jugador1Vect_J1Vect{4,6}" : Int = PLC Jugador1Vect.J1Vect[4,6] AT %DB4.DBW84, 1 s
   "Jugador1Vect_J1Vect{4,7}" : Int = PLC Jugador1Vect.J1Vect[4,7] AT %DB4.DBW86, 1 s
   "Jugador1Vect_J1Vect{4,8}" : Int = PLC Jugador1Vect.J1Vect[4,8] AT %DB4.DBW88, 1 s
   "Jugador1Vect_J1Vect{5,0}" : Int = PLC Jugador1Vect.J1Vect[5,0] AT %DB4.DBW90, 1 s
   "Jugador1Vect_J1Vect{5,1}" : Int = PLC Jugador1Vect.J1Vect[5,1] AT %DB4.DBW92, 1 s
   "Jugador1Vect_J1Vect{5,2}" : Int = PLC Jugador1Vect.J1Vect[5,2] AT %DB4.DBW94, 1 s
   "Jugador1Vect_J1Vect{5,3}" : Int = PLC Jugador1Vect.J1Vect[5,3] AT %DB4.DBW96, 1 s
   "Jugador1Vect_J1Vect{5,4}" : Int = PLC Jugador1Vect.J1Vect[5,4] AT %DB4.DBW98, 1 s
   "Jugador1Vect_J1Vect{5,5}" : Int = PLC Jugador1Vect.J1Vect[5,5] AT %DB4.DBW100, 1 s
   "Jugador1Vect_J1Vect{5,6}" : Int = PLC Jugador1Vect.J1Vect[5,6] AT %DB4.DBW102, 1 s
   "Jugador1Vect_J1Vect{5,7}" : Int = PLC Jugador1Vect.J1Vect[5,7] AT %DB4.DBW104, 1 s
   "Jugador1Vect_J1Vect{5,8}" : Int = PLC Jugador1Vect.J1Vect[5,8] AT %DB4.DBW106, 1 s
   "Jugador1Vect_J1Vect{6,0}" : Int = PLC Jugador1Vect.J1Vect[6,0] AT %DB4.DBW108, 1 s
   "Jugador1Vect_J1Vect{6,1}" : Int = PLC Jugador1Vect.J1Vect[6,1] AT %DB4.DBW110, 1 s
   "Jugador1Vect_J1Vect{6,2}" : Int = PLC Jugador1Vect.J1Vect[6,2] AT %DB4.DBW112, 1 s
   "Jugador1Vect_J1Vect{6,3}" : Int = PLC Jugador1Vect.J1Vect[6,3] AT %DB4.DBW114, 1 s
   "Jugador1Vect_J1Vect{6,4}" : Int = PLC Jugador1Vect.J1Vect[6,4] AT %DB4.DBW116, 1 s
   "Jugador1Vect_J1Vect{6,5}" : Int = PLC Jugador1Vect.J1Vect[6,5] AT %DB4.DBW118, 1 s
   "Jugador1Vect_J1Vect{6,6}" : Int = PLC Jugador1Vect.J1Vect[6,6] AT %DB4.DBW120, 1 s
   "Jugador1Vect_J1Vect{6,7}" : Int = PLC Jugador1Vect.J1Vect[6,7] AT %DB4.DBW122, 1 s
   "Jugador1Vect_J1Vect{6,8}" : Int = PLC Jugador1Vect.J1Vect[6,8] AT %DB4.DBW124, 1 s
   "Jugador1Vect_J1Vect{7,0}" : Int = PLC Jugador1Vect.J1Vect[7,0] AT %DB4.DBW126, 1 s
   "Jugador1Vect_J1Vect{7,1}" : Int = PLC Jugador1Vect.J1Vect[7,1] AT %DB4.DBW128, 1 s
   "Jugador1Vect_J1Vect{7,2}" : Int = PLC Jugador1Vect.J1Vect[7,2] AT %DB4.DBW130, 1 s
   "Jugador1Vect_J1Vect{7,3}" : Int = PLC Jugador1Vect.J1Vect[7,3] AT %DB4.DBW132, 1 s
   "Jugador1Vect_J1Vect{7,4}" : Int = PLC Jugador1Vect.J1Vect[7,4] AT %DB4.DBW134, 1 s
   "Jugador1Vect_J1Vect{7,5}" : Int = PLC Jugador1Vect.J1Vect[7,5] AT %DB4.DBW136, 1 s
   "Jugador1Vect_J1Vect{7,6}" : Int = PLC Jugador1Vect.J1Vect[7,6] AT %DB4.DBW138, 1 s
   "Jugador1Vect_J1Vect{7,7}" : Int = PLC Jugador1Vect.J1Vect[7,7] AT %DB4.DBW140, 1 s
   "Jugador1Vect_J1Vect{7,8}" : Int = PLC Jugador1Vect.J1Vect[7,8] AT %DB4.DBW142, 1 s
   "ReiniciarJ1" : Bool = PLC ReiniciarJ1 AT %M13.1, 1 s
   "Conecta4J1" : Bool = PLC Conecta4J1 AT %M13.2, 1 s
   "Conecta5J1" : Bool = PLC Conecta5J1 AT %M13.3, 1 s
   "ResetJ1Send" : Bool = PLC ResetJ1Send AT %M18.0, 1 s
   "ResetJ2Rec" : Bool = PLC ResetJ2Rec AT %M18.1, 1 s

screen "Root screen" 800x420, template "Template_1"
   on GenerateScreen: SetTag("Tag_ScreenNumber", 1)
   Button "Button_3" at 132,28 size 26x27; TextOff 'Text'
      Visibility <- "PanelJ1"
      on Press: SetBit("B1J1")
      on Release: ResetBit("B1J1")
   Button "Button_1" at 160,28 size 26x27; TextOff 'Text'
      Visibility <- "PanelJ1"
      on Press: SetBit("B2J1")
      on Release: ResetBit("B2J1")
   Button "Button_2" at 187,28 size 26x27; TextOff 'Text'
      Visibility <- "PanelJ1"
      on Press: SetBit("B3J1")
      on Release: ResetBit("B3J1")
   Button "Button_4" at 213,28 size 26x27; TextOff 'Text'
      Visibility <- "PanelJ1"
      on Press: SetBit("B4J1")
      on Release: ResetBit("B4J1")
   Button "Button_5" at 240,28 size 26x27; TextOff 'Text'
      Visibility <- "PanelJ1"
      on Press: SetBit("B5J1")
      on Release: ResetBit("B5J1")
   Button "Button_6" at 268,28 size 26x27; TextOff 'Text'
      Visibility <- "PanelJ1"
      on Press: SetBit("B6J1")
      on Release: ResetBit("B6J1")
   Button "Button_7" at 295,28 size 26x27; TextOff 'Text'
      Visibility <- "PanelJ1"
      on Press: ResetBit("B7J1")
      on Release: ResetBit("B7J1")
   Button "Button_8" at 321,28 size 26x27; TextOff 'Text'
      Visibility <- "PanelJ1"
      on Press: SetBit("B8J1")
      on Release: ResetBit("B8J1")
   Button "Button_9" at 348,28 size 26x27; TextOff 'Text'
      Visibility <- "PanelJ1"
      on Press: SetBit("B9J1")
      on Release: ResetBit("B9J1")
   Button "Button_10" at 512,18 size 169x40; TextOff 'Reiniciar Juego'
      on Press: SetBit("ReiniciarJ1")
      on Release: ResetBit("ReiniciarJ1")
   TextField "Text field_1" at 456,64 size 295x23; Text '1. Selecciona el Modo de Juego:'
   TextField "Text field_2" at 470,139 size 264x23; Text 'Modo de Juego Seleccionado'
      Visibility <- "Mensaje1J1"
   TextField "Text field_3" at 479,167 size 270x23; Text 'MODO CONECTA 4 ACTIVADO'
      Visibility <- "Mensaje2J1"
   TextField "Text field_4" at 481,167 size 270x23; Text 'MODO CONECTA 5 ACTIVADO'
      Visibility <- "Mensaje3J1"
   TextField "Text field_5" at 446,193 size 303x42; Text 'ES TU TURNO (Selecciona una Columna Valida)'
      Visibility <- "Mensaje4J1"
   TextField "Text field_6" at 479,236 size 235x42; Text 'TURNO DE TU OPONENTE (Espera)'
      Visibility <- "Mensaje5J1"
   TextField "Text field_7" at 464,291 size 109x23; Text 'GANASTE!!!'
      Visibility <- "Mensaje6J1"
   TextField "Text field_8" at 617,291 size 117x23; Text 'PERDISTE :('
      Visibility <- "Mensaje7J1"
   Button "Button_11" at 481,96 size 104x40; TextOff 'Conecta 4'
      on Press: SetBit("Conecta4J1")
      on Release: ResetBit("Conecta4J1")
   Button "Button_12" at 594,95 size 104x40; TextOff 'Conecta 5'
      on Press: SetBit("Conecta5J1")
      on Release: ResetBit("Conecta5J1")
   Circle "Circle_1" at 131,99 size 27x27
      Appearance <- "Jugador1Vect_J1Vect{7,0}"
   Circle "Circle_2" at 158,99 size 27x27
      Appearance <- "Jugador1Vect_J1Vect{7,1}"
   Circle "Circle_3" at 185,99 size 27x27
      Appearance <- "Jugador1Vect_J1Vect{7,2}"
   Circle "Circle_4" at 212,99 size 27x27
      Appearance <- "Jugador1Vect_J1Vect{7,3}"
   Circle "Circle_5" at 239,99 size 27x27
      Appearance <- "Jugador1Vect_J1Vect{7,4}"
   Circle "Circle_6" at 266,99 size 27x27
      Appearance <- "Jugador1Vect_J1Vect{7,5}"
   Circle "Circle_7" at 293,99 size 27x27
      Appearance <- "Jugador1Vect_J1Vect{7,6}"
   Circle "Circle_8" at 320,99 size 27x27
      Appearance <- "Jugador1Vect_J1Vect{7,7}"
   Circle "Circle_9" at 347,99 size 27x27
      Appearance <- "Jugador1Vect_J1Vect{7,8}"
   Circle "Circle_10" at 131,126 size 27x27
      Appearance <- "Jugador1Vect_J1Vect{6,0}"
   Circle "Circle_11" at 158,126 size 27x27
      Appearance <- "Jugador1Vect_J1Vect{6,1}"
   Circle "Circle_12" at 185,126 size 27x27
      Appearance <- "Jugador1Vect_J1Vect{6,2}"
   Circle "Circle_13" at 212,126 size 27x27
      Appearance <- "Jugador1Vect_J1Vect{6,3}"
   Circle "Circle_14" at 239,126 size 27x27
      Appearance <- "Jugador1Vect_J1Vect{6,4}"
   Circle "Circle_15" at 266,126 size 27x27
      Appearance <- "Jugador1Vect_J1Vect{6,5}"
   Circle "Circle_16" at 293,126 size 27x27
      Appearance <- "Jugador1Vect_J1Vect{6,6}"
   Circle "Circle_17" at 320,126 size 27x27
      Appearance <- "Jugador1Vect_J1Vect{6,7}"
   Circle "Circle_18" at 347,126 size 27x27
      Appearance <- "Jugador1Vect_J1Vect{6,8}"
   Circle "Circle_19" at 131,153 size 27x27
      Appearance <- "Jugador1Vect_J1Vect{5,0}"
   Circle "Circle_20" at 158,153 size 27x27
      Appearance <- "Jugador1Vect_J1Vect{5,1}"
   Circle "Circle_21" at 185,153 size 27x27
      Appearance <- "Jugador1Vect_J1Vect{5,2}"
   Circle "Circle_22" at 212,153 size 27x27
      Appearance <- "Jugador1Vect_J1Vect{5,3}"
   Circle "Circle_23" at 239,153 size 27x27
      Appearance <- "Jugador1Vect_J1Vect{5,4}"
   Circle "Circle_24" at 266,153 size 27x27
      Appearance <- "Jugador1Vect_J1Vect{5,5}"
   Circle "Circle_25" at 293,153 size 27x27
      Appearance <- "Jugador1Vect_J1Vect{5,6}"
   Circle "Circle_26" at 320,153 size 27x27
      Appearance <- "Jugador1Vect_J1Vect{5,7}"
   Circle "Circle_27" at 347,153 size 27x27
      Appearance <- "Jugador1Vect_J1Vect{5,8}"
   Circle "Circle_28" at 131,180 size 27x27
      Appearance <- "Jugador1Vect_J1Vect{4,0}"
   Circle "Circle_29" at 158,180 size 27x27
      Appearance <- "Jugador1Vect_J1Vect{4,1}"
   Circle "Circle_30" at 185,180 size 27x27
      Appearance <- "Jugador1Vect_J1Vect{4,2}"
   Circle "Circle_31" at 212,180 size 27x27
      Appearance <- "Jugador1Vect_J1Vect{4,3}"
   Circle "Circle_32" at 239,180 size 27x27
      Appearance <- "Jugador1Vect_J1Vect{4,4}"
   Circle "Circle_33" at 266,180 size 27x27
      Appearance <- "Jugador1Vect_J1Vect{4,5}"
   Circle "Circle_34" at 293,180 size 27x27
      Appearance <- "Jugador1Vect_J1Vect{4,6}"
   Circle "Circle_35" at 320,180 size 27x27
      Appearance <- "Jugador1Vect_J1Vect{4,7}"
   Circle "Circle_36" at 347,180 size 27x27
      Appearance <- "Jugador1Vect_J1Vect{4,8}"
   Circle "Circle_37" at 131,207 size 27x27
      Appearance <- "Jugador1Vect_J1Vect{3,0}"
   Circle "Circle_38" at 158,207 size 27x27
      Appearance <- "Jugador1Vect_J1Vect{3,1}"
   Circle "Circle_39" at 185,207 size 27x27
      Appearance <- "Jugador1Vect_J1Vect{3,2}"
   Circle "Circle_40" at 212,207 size 27x27
      Appearance <- "Jugador1Vect_J1Vect{3,3}"
   Circle "Circle_41" at 239,207 size 27x27
      Appearance <- "Jugador1Vect_J1Vect{3,4}"
   Circle "Circle_42" at 266,207 size 27x27
      Appearance <- "Jugador1Vect_J1Vect{3,5}"
   Circle "Circle_43" at 293,207 size 27x27
      Appearance <- "Jugador1Vect_J1Vect{3,6}"
   Circle "Circle_44" at 320,207 size 27x27
      Appearance <- "Jugador1Vect_J1Vect{3,7}"
   Circle "Circle_45" at 347,207 size 27x27
      Appearance <- "Jugador1Vect_J1Vect{3,8}"
   Circle "Circle_46" at 131,234 size 27x27
      Appearance <- "Jugador1Vect_J1Vect{2,0}"
   Circle "Circle_47" at 158,234 size 27x27
      Appearance <- "Jugador1Vect_J1Vect{2,1}"
   Circle "Circle_48" at 185,234 size 27x27
      Appearance <- "Jugador1Vect_J1Vect{2,2}"
   Circle "Circle_49" at 212,234 size 27x27
      Appearance <- "Jugador1Vect_J1Vect{2,3}"
   Circle "Circle_50" at 239,234 size 27x27
      Appearance <- "Jugador1Vect_J1Vect{2,4}"
   Circle "Circle_51" at 266,234 size 27x27
      Appearance <- "Jugador1Vect_J1Vect{2,5}"
   Circle "Circle_52" at 293,234 size 27x27
      Appearance <- "Jugador1Vect_J1Vect{2,6}"
   Circle "Circle_53" at 320,234 size 27x27
      Appearance <- "Jugador1Vect_J1Vect{2,7}"
   Circle "Circle_54" at 347,234 size 27x27
      Appearance <- "Jugador1Vect_J1Vect{2,8}"
   Circle "Circle_55" at 131,261 size 27x27
      Appearance <- "Jugador1Vect_J1Vect{1,0}"
   Circle "Circle_56" at 158,261 size 27x27
      Appearance <- "Jugador1Vect_J1Vect{1,1}"
   Circle "Circle_57" at 185,261 size 27x27
      Appearance <- "Jugador1Vect_J1Vect{1,2}"
   Circle "Circle_58" at 212,261 size 27x27
      Appearance <- "Jugador1Vect_J1Vect{1,3}"
   Circle "Circle_59" at 239,261 size 27x27
      Appearance <- "Jugador1Vect_J1Vect{1,4}"
   Circle "Circle_60" at 266,261 size 27x27
      Appearance <- "Jugador1Vect_J1Vect{1,5}"
   Circle "Circle_61" at 293,261 size 27x27
      Appearance <- "Jugador1Vect_J1Vect{1,6}"
   Circle "Circle_62" at 320,261 size 27x27
      Appearance <- "Jugador1Vect_J1Vect{1,7}"
   Circle "Circle_63" at 347,261 size 27x27
      Appearance <- "Jugador1Vect_J1Vect{1,8}"
   TextField "Text field_9" at 3,25 size 129x40; Text 'JUGADOR 1 FICHAS ROJAS'
   Circle "Circle_64" at 131,288 size 27x27
      Appearance <- "Jugador1Vect_J1Vect{0,0}"
   Circle "Circle_65" at 159,288 size 27x27
      Appearance <- "Jugador1Vect_J1Vect{0,1}"
   Circle "Circle_66" at 186,288 size 27x27
      Appearance <- "Jugador1Vect_J1Vect{0,2}"
   Circle "Circle_67" at 213,288 size 27x27
      Appearance <- "Jugador1Vect_J1Vect{0,3}"
   Circle "Circle_68" at 240,288 size 27x27
      Appearance <- "Jugador1Vect_J1Vect{0,4}"
   Circle "Circle_69" at 267,288 size 27x27
      Appearance <- "Jugador1Vect_J1Vect{0,5}"
   Circle "Circle_70" at 294,288 size 27x27
      Appearance <- "Jugador1Vect_J1Vect{0,6}"
   Circle "Circle_71" at 321,288 size 27x27
      Appearance <- "Jugador1Vect_J1Vect{0,7}"
   Circle "Circle_72" at 348,288 size 27x27
      Appearance <- "Jugador1Vect_J1Vect{0,8}"

Template "Template_1" 800x420
   Button "Exit" at 720,360 size 78x58; TextOff 'Exit'; PictureOff "ExitRuntime_TP700_Comfort_TR"; PictureOn "ExitRuntime_TP700_Comfort_TR"
      on Release: StopRuntime(0)
   Button "Template_Button" at 640,360 size 78x58; TextOff 'Text'
   Button "Template_Button_1" at 560,360 size 78x58; TextOff 'Text'
   Button "Template_Button_2" at 480,360 size 78x58; TextOff 'Text'
   Button "Template_Button_3" at 400,360 size 78x58; TextOff 'Text'
   Button "Template_Button_4" at 321,360 size 78x58; TextOff 'Text'
   Button "Template_Button_5" at 241,360 size 78x58; TextOff 'Text'
   Button "Template_Button_6" at 161,360 size 78x58; TextOff 'Text'
   Button "Alarms" at 81,360 size 78x58; TextOff 'Alarms'; PictureOff "AlarmDisplay_TP700_Comfort_TR"; PictureOn "AlarmDisplay_TP700_Comfort_TR"
      on Release: function_ef3f5d25("Alarm window_Unacknowledged", -1)
   Button "Start screen" at 1,360 size 78x58; TextOff 'Start screen'; PictureOff "NavigateHome_TP700_Comfort_TR"; PictureOn "NavigateHome_TP700_Comfort_TR"
      on Release: ActivateScreen("Root screen", 0)
*)

(* ===== HMI "HMI_RT_2" =====
system functions are stored by id; their names below are inferred from use
connection "HMI_Connection_2": ETHERNET, S7_1500_OMS

HMI tags "Default tag table"
   "Tag_ScreenNumber" : UInt, internal
   "Mensaje1J2" : Bool = PLC Mensaje1J2 AT %M11.0, 1 s
   "Mensaje2J2" : Bool = PLC Mensaje2J2 AT %M11.1, 1 s
   "Mensaje3J2" : Bool = PLC Mensaje3J2 AT %M11.2, 1 s
   "Mensaje4J2" : Bool = PLC Mensaje4J2 AT %M11.3, 1 s
   "Mensaje5J2" : Bool = PLC Mensaje5J2 AT %M11.4, 1 s
   "Mensaje6J2" : Bool = PLC Mensaje6J2 AT %M11.5, 1 s
   "Mensaje7J2" : Bool = PLC Mensaje7J2 AT %M11.6, 1 s
   "PanelJ2" : Bool = PLC PanelJ2 AT %M13.0, 1 s
   "B1J2" : Bool = PLC B1J2 AT %M11.7, 1 s
   "B2J2" : Bool = PLC B2J2 AT %M12.0, 1 s
   "B3J2" : Bool = PLC B3J2 AT %M12.1, 1 s
   "B4J2" : Bool = PLC B4J2 AT %M12.2, 1 s
   "B5J2" : Bool = PLC B5J2 AT %M12.3, 1 s
   "B6J2" : Bool = PLC B6J2 AT %M12.4, 1 s
   "B7J2" : Bool = PLC B7J2 AT %M12.5, 1 s
   "B8J2" : Bool = PLC B8J2 AT %M12.6, 1 s
   "B9J2" : Bool = PLC B9J2 AT %M12.7, 1 s
   "ReiniciarJ2" : Bool = PLC ReiniciarJ2 AT %M13.1, 1 s
   "Conecta4J2" : Bool = PLC Conecta4J2 AT %M13.2, 1 s
   "Conecta5J2" : Bool = PLC Conecta5J2 AT %M13.3, 1 s
   "Jugador2Vect_J2Vect{0,0}" : Int = PLC Jugador2Vect.J2Vect[0,0] AT %DB4.DBW0, 1 s
   "Jugador2Vect_J2Vect{0,1}" : Int = PLC Jugador2Vect.J2Vect[0,1] AT %DB4.DBW2, 1 s
   "Jugador2Vect_J2Vect{0,2}" : Int = PLC Jugador2Vect.J2Vect[0,2] AT %DB4.DBW4, 1 s
   "Jugador2Vect_J2Vect{0,3}" : Int = PLC Jugador2Vect.J2Vect[0,3] AT %DB4.DBW6, 1 s
   "Jugador2Vect_J2Vect{0,4}" : Int = PLC Jugador2Vect.J2Vect[0,4] AT %DB4.DBW8, 1 s
   "Jugador2Vect_J2Vect{0,5}" : Int = PLC Jugador2Vect.J2Vect[0,5] AT %DB4.DBW10, 1 s
   "Jugador2Vect_J2Vect{0,6}" : Int = PLC Jugador2Vect.J2Vect[0,6] AT %DB4.DBW12, 1 s
   "Jugador2Vect_J2Vect{0,7}" : Int = PLC Jugador2Vect.J2Vect[0,7] AT %DB4.DBW14, 1 s
   "Jugador2Vect_J2Vect{0,8}" : Int = PLC Jugador2Vect.J2Vect[0,8] AT %DB4.DBW16, 1 s
   "Jugador2Vect_J2Vect{1,0}" : Int = PLC Jugador2Vect.J2Vect[1,0] AT %DB4.DBW18, 1 s
   "Jugador2Vect_J2Vect{1,1}" : Int = PLC Jugador2Vect.J2Vect[1,1] AT %DB4.DBW20, 1 s
   "Jugador2Vect_J2Vect{1,2}" : Int = PLC Jugador2Vect.J2Vect[1,2] AT %DB4.DBW22, 1 s
   "Jugador2Vect_J2Vect{1,3}" : Int = PLC Jugador2Vect.J2Vect[1,3] AT %DB4.DBW24, 1 s
   "Jugador2Vect_J2Vect{1,4}" : Int = PLC Jugador2Vect.J2Vect[1,4] AT %DB4.DBW26, 1 s
   "Jugador2Vect_J2Vect{1,5}" : Int = PLC Jugador2Vect.J2Vect[1,5] AT %DB4.DBW28, 1 s
   "Jugador2Vect_J2Vect{1,6}" : Int = PLC Jugador2Vect.J2Vect[1,6] AT %DB4.DBW30, 1 s
   "Jugador2Vect_J2Vect{1,7}" : Int = PLC Jugador2Vect.J2Vect[1,7] AT %DB4.DBW32, 1 s
   "Jugador2Vect_J2Vect{1,8}" : Int = PLC Jugador2Vect.J2Vect[1,8] AT %DB4.DBW34, 1 s
   "Jugador2Vect_J2Vect{2,0}" : Int = PLC Jugador2Vect.J2Vect[2,0] AT %DB4.DBW36, 1 s
   "Jugador2Vect_J2Vect{2,1}" : Int = PLC Jugador2Vect.J2Vect[2,1] AT %DB4.DBW38, 1 s
   "Jugador2Vect_J2Vect{2,2}" : Int = PLC Jugador2Vect.J2Vect[2,2] AT %DB4.DBW40, 1 s
   "Jugador2Vect_J2Vect{2,3}" : Int = PLC Jugador2Vect.J2Vect[2,3] AT %DB4.DBW42, 1 s
   "Jugador2Vect_J2Vect{2,4}" : Int = PLC Jugador2Vect.J2Vect[2,4] AT %DB4.DBW44, 1 s
   "Jugador2Vect_J2Vect{2,5}" : Int = PLC Jugador2Vect.J2Vect[2,5] AT %DB4.DBW46, 1 s
   "Jugador2Vect_J2Vect{2,6}" : Int = PLC Jugador2Vect.J2Vect[2,6] AT %DB4.DBW48, 1 s
   "Jugador2Vect_J2Vect{2,7}" : Int = PLC Jugador2Vect.J2Vect[2,7] AT %DB4.DBW50, 1 s
   "Jugador2Vect_J2Vect{2,8}" : Int = PLC Jugador2Vect.J2Vect[2,8] AT %DB4.DBW52, 1 s
   "Jugador2Vect_J2Vect{3,0}" : Int = PLC Jugador2Vect.J2Vect[3,0] AT %DB4.DBW54, 1 s
   "Jugador2Vect_J2Vect{3,1}" : Int = PLC Jugador2Vect.J2Vect[3,1] AT %DB4.DBW56, 1 s
   "Jugador2Vect_J2Vect{3,2}" : Int = PLC Jugador2Vect.J2Vect[3,2] AT %DB4.DBW58, 1 s
   "Jugador2Vect_J2Vect{3,3}" : Int = PLC Jugador2Vect.J2Vect[3,3] AT %DB4.DBW60, 1 s
   "Jugador2Vect_J2Vect{3,4}" : Int = PLC Jugador2Vect.J2Vect[3,4] AT %DB4.DBW62, 1 s
   "Jugador2Vect_J2Vect{3,5}" : Int = PLC Jugador2Vect.J2Vect[3,5] AT %DB4.DBW64, 1 s
   "Jugador2Vect_J2Vect{3,6}" : Int = PLC Jugador2Vect.J2Vect[3,6] AT %DB4.DBW66, 1 s
   "Jugador2Vect_J2Vect{3,7}" : Int = PLC Jugador2Vect.J2Vect[3,7] AT %DB4.DBW68, 1 s
   "Jugador2Vect_J2Vect{3,8}" : Int = PLC Jugador2Vect.J2Vect[3,8] AT %DB4.DBW70, 1 s
   "Jugador2Vect_J2Vect{4,0}" : Int = PLC Jugador2Vect.J2Vect[4,0] AT %DB4.DBW72, 1 s
   "Jugador2Vect_J2Vect{4,1}" : Int = PLC Jugador2Vect.J2Vect[4,1] AT %DB4.DBW74, 1 s
   "Jugador2Vect_J2Vect{4,2}" : Int = PLC Jugador2Vect.J2Vect[4,2] AT %DB4.DBW76, 1 s
   "Jugador2Vect_J2Vect{4,3}" : Int = PLC Jugador2Vect.J2Vect[4,3] AT %DB4.DBW78, 1 s
   "Jugador2Vect_J2Vect{4,4}" : Int = PLC Jugador2Vect.J2Vect[4,4] AT %DB4.DBW80, 1 s
   "Jugador2Vect_J2Vect{4,5}" : Int = PLC Jugador2Vect.J2Vect[4,5] AT %DB4.DBW82, 1 s
   "Jugador2Vect_J2Vect{4,6}" : Int = PLC Jugador2Vect.J2Vect[4,6] AT %DB4.DBW84, 1 s
   "Jugador2Vect_J2Vect{4,7}" : Int = PLC Jugador2Vect.J2Vect[4,7] AT %DB4.DBW86, 1 s
   "Jugador2Vect_J2Vect{4,8}" : Int = PLC Jugador2Vect.J2Vect[4,8] AT %DB4.DBW88, 1 s
   "Jugador2Vect_J2Vect{5,0}" : Int = PLC Jugador2Vect.J2Vect[5,0] AT %DB4.DBW90, 1 s
   "Jugador2Vect_J2Vect{5,1}" : Int = PLC Jugador2Vect.J2Vect[5,1] AT %DB4.DBW92, 1 s
   "Jugador2Vect_J2Vect{5,2}" : Int = PLC Jugador2Vect.J2Vect[5,2] AT %DB4.DBW94, 1 s
   "Jugador2Vect_J2Vect{5,3}" : Int = PLC Jugador2Vect.J2Vect[5,3] AT %DB4.DBW96, 1 s
   "Jugador2Vect_J2Vect{5,4}" : Int = PLC Jugador2Vect.J2Vect[5,4] AT %DB4.DBW98, 1 s
   "Jugador2Vect_J2Vect{5,5}" : Int = PLC Jugador2Vect.J2Vect[5,5] AT %DB4.DBW100, 1 s
   "Jugador2Vect_J2Vect{5,6}" : Int = PLC Jugador2Vect.J2Vect[5,6] AT %DB4.DBW102, 1 s
   "Jugador2Vect_J2Vect{5,7}" : Int = PLC Jugador2Vect.J2Vect[5,7] AT %DB4.DBW104, 1 s
   "Jugador2Vect_J2Vect{5,8}" : Int = PLC Jugador2Vect.J2Vect[5,8] AT %DB4.DBW106, 1 s
   "Jugador2Vect_J2Vect{6,0}" : Int = PLC Jugador2Vect.J2Vect[6,0] AT %DB4.DBW108, 1 s
   "Jugador2Vect_J2Vect{6,1}" : Int = PLC Jugador2Vect.J2Vect[6,1] AT %DB4.DBW110, 1 s
   "Jugador2Vect_J2Vect{6,2}" : Int = PLC Jugador2Vect.J2Vect[6,2] AT %DB4.DBW112, 1 s
   "Jugador2Vect_J2Vect{6,3}" : Int = PLC Jugador2Vect.J2Vect[6,3] AT %DB4.DBW114, 1 s
   "Jugador2Vect_J2Vect{6,4}" : Int = PLC Jugador2Vect.J2Vect[6,4] AT %DB4.DBW116, 1 s
   "Jugador2Vect_J2Vect{6,5}" : Int = PLC Jugador2Vect.J2Vect[6,5] AT %DB4.DBW118, 1 s
   "Jugador2Vect_J2Vect{6,6}" : Int = PLC Jugador2Vect.J2Vect[6,6] AT %DB4.DBW120, 1 s
   "Jugador2Vect_J2Vect{6,7}" : Int = PLC Jugador2Vect.J2Vect[6,7] AT %DB4.DBW122, 1 s
   "Jugador2Vect_J2Vect{6,8}" : Int = PLC Jugador2Vect.J2Vect[6,8] AT %DB4.DBW124, 1 s
   "Jugador2Vect_J2Vect{7,0}" : Int = PLC Jugador2Vect.J2Vect[7,0] AT %DB4.DBW126, 1 s
   "Jugador2Vect_J2Vect{7,1}" : Int = PLC Jugador2Vect.J2Vect[7,1] AT %DB4.DBW128, 1 s
   "Jugador2Vect_J2Vect{7,2}" : Int = PLC Jugador2Vect.J2Vect[7,2] AT %DB4.DBW130, 1 s
   "Jugador2Vect_J2Vect{7,3}" : Int = PLC Jugador2Vect.J2Vect[7,3] AT %DB4.DBW132, 1 s
   "Jugador2Vect_J2Vect{7,4}" : Int = PLC Jugador2Vect.J2Vect[7,4] AT %DB4.DBW134, 1 s
   "Jugador2Vect_J2Vect{7,5}" : Int = PLC Jugador2Vect.J2Vect[7,5] AT %DB4.DBW136, 1 s
   "Jugador2Vect_J2Vect{7,6}" : Int = PLC Jugador2Vect.J2Vect[7,6] AT %DB4.DBW138, 1 s
   "Jugador2Vect_J2Vect{7,7}" : Int = PLC Jugador2Vect.J2Vect[7,7] AT %DB4.DBW140, 1 s
   "Jugador2Vect_J2Vect{7,8}" : Int = PLC Jugador2Vect.J2Vect[7,8] AT %DB4.DBW142, 1 s

screen "Root screen" 800x420, template "Template_1"
   on GenerateScreen: SetTag("Tag_ScreenNumber", 1)
   Button "Button_3" at 140,28 size 26x27; TextOff 'Text'
      Visibility <- "PanelJ2"
      on Press: SetBit("B1J2")
      on Release: ResetBit("B1J2")
   Button "Button_1" at 168,28 size 26x27; TextOff 'Text'
      Visibility <- "PanelJ2"
      on Press: SetBit("B2J2")
      on Release: ResetBit("B2J2")
   Button "Button_2" at 195,28 size 26x27; TextOff 'Text'
      Visibility <- "PanelJ2"
      on Press: SetBit("B3J2")
      on Release: ResetBit("B3J2")
   Button "Button_4" at 221,28 size 26x27; TextOff 'Text'
      Visibility <- "PanelJ2"
      on Press: SetBit("B4J2")
      on Release: ResetBit("B4J2")
   Button "Button_5" at 248,28 size 26x27; TextOff 'Text'
      Visibility <- "PanelJ2"
      on Press: SetBit("B5J2")
      on Release: ResetBit("B5J2")
   Button "Button_6" at 276,28 size 26x27; TextOff 'Text'
      Visibility <- "PanelJ2"
      on Press: SetBit("B6J2")
      on Release: ResetBit("B6J2")
   Button "Button_7" at 303,28 size 26x27; TextOff 'Text'
      Visibility <- "PanelJ2"
      on Press: SetBit("B7J2")
      on Release: ResetBit("B7J2")
   Button "Button_8" at 329,28 size 26x27; TextOff 'Text'
      Visibility <- "PanelJ2"
      on Press: SetBit("B8J2")
      on Release: ResetBit("B8J2")
   Button "Button_9" at 356,28 size 26x27; TextOff 'Text'
      Visibility <- "PanelJ2"
      on Press: SetBit("B9J2")
      on Release: ResetBit("B9J2")
   TextField "Text field_3" at 481,94 size 270x23; Text 'MODO CONECTA 4 ACTIVADO'
      Visibility <- "Mensaje2J2"
   TextField "Text field_4" at 481,95 size 270x23; Text 'MODO CONECTA 5 ACTIVADO'
      Visibility <- "Mensaje3J2"
   TextField "Text field_5" at 452,138 size 303x42; Text 'ES TU TURNO (Selecciona una Columna Valida)'
      Visibility <- "Mensaje4J2"
   TextField "Text field_6" at 481,207 size 235x42; Text 'TURNO DE TU OPONENTE (Espera)'
      Visibility <- "Mensaje5J2"
   TextField "Text field_7" at 467,278 size 109x23; Text 'GANASTE!!!'
      Visibility <- "Mensaje6J2"
   TextField "Text field_8" at 622,278 size 117x23; Text 'PERDISTE :('
      Visibility <- "Mensaje7J2"
   Circle "Circle_1" at 139,99 size 27x27
      Appearance <- "Jugador2Vect_J2Vect{7,0}"
   Circle "Circle_2" at 166,99 size 27x27
      Appearance <- "Jugador2Vect_J2Vect{7,1}"
   Circle "Circle_3" at 193,99 size 27x27
      Appearance <- "Jugador2Vect_J2Vect{7,2}"
   Circle "Circle_4" at 220,99 size 27x27
      Appearance <- "Jugador2Vect_J2Vect{7,3}"
   Circle "Circle_5" at 247,99 size 27x27
      Appearance <- "Jugador2Vect_J2Vect{7,4}"
   Circle "Circle_6" at 274,99 size 27x27
      Appearance <- "Jugador2Vect_J2Vect{7,5}"
   Circle "Circle_7" at 301,99 size 27x27
      Appearance <- "Jugador2Vect_J2Vect{7,6}"
   Circle "Circle_8" at 328,99 size 27x27
      Appearance <- "Jugador2Vect_J2Vect{7,7}"
   Circle "Circle_9" at 355,99 size 27x27
      Appearance <- "Jugador2Vect_J2Vect{7,8}"
   Circle "Circle_10" at 139,126 size 27x27
      Appearance <- "Jugador2Vect_J2Vect{6,0}"
   Circle "Circle_11" at 166,126 size 27x27
      Appearance <- "Jugador2Vect_J2Vect{6,1}"
   Circle "Circle_12" at 193,126 size 27x27
      Appearance <- "Jugador2Vect_J2Vect{6,2}"
   Circle "Circle_13" at 220,126 size 27x27
      Appearance <- "Jugador2Vect_J2Vect{6,3}"
   Circle "Circle_14" at 247,126 size 27x27
      Appearance <- "Jugador2Vect_J2Vect{6,4}"
   Circle "Circle_15" at 274,126 size 27x27
      Appearance <- "Jugador2Vect_J2Vect{6,5}"
   Circle "Circle_16" at 301,126 size 27x27
      Appearance <- "Jugador2Vect_J2Vect{6,6}"
   Circle "Circle_17" at 328,126 size 27x27
      Appearance <- "Jugador2Vect_J2Vect{6,7}"
   Circle "Circle_18" at 355,126 size 27x27
      Appearance <- "Jugador2Vect_J2Vect{6,8}"
   Circle "Circle_19" at 139,153 size 27x27
      Appearance <- "Jugador2Vect_J2Vect{5,0}"
   Circle "Circle_20" at 166,153 size 27x27
      Appearance <- "Jugador2Vect_J2Vect{5,1}"
   Circle "Circle_21" at 193,153 size 27x27
      Appearance <- "Jugador2Vect_J2Vect{5,2}"
   Circle "Circle_22" at 220,153 size 27x27
      Appearance <- "Jugador2Vect_J2Vect{5,3}"
   Circle "Circle_23" at 247,153 size 27x27
      Appearance <- "Jugador2Vect_J2Vect{5,4}"
   Circle "Circle_24" at 274,153 size 27x27
      Appearance <- "Jugador2Vect_J2Vect{5,5}"
   Circle "Circle_25" at 301,153 size 27x27
      Appearance <- "Jugador2Vect_J2Vect{5,6}"
   Circle "Circle_26" at 328,153 size 27x27
      Appearance <- "Jugador2Vect_J2Vect{5,7}"
   Circle "Circle_27" at 355,153 size 27x27
      Appearance <- "Jugador2Vect_J2Vect{5,8}"
   Circle "Circle_28" at 139,180 size 27x27
      Appearance <- "Jugador2Vect_J2Vect{4,0}"
   Circle "Circle_29" at 166,180 size 27x27
      Appearance <- "Jugador2Vect_J2Vect{4,1}"
   Circle "Circle_30" at 193,180 size 27x27
      Appearance <- "Jugador2Vect_J2Vect{4,2}"
   Circle "Circle_31" at 220,180 size 27x27
      Appearance <- "Jugador2Vect_J2Vect{4,3}"
   Circle "Circle_32" at 247,180 size 27x27
      Appearance <- "Jugador2Vect_J2Vect{4,4}"
   Circle "Circle_33" at 274,180 size 27x27
      Appearance <- "Jugador2Vect_J2Vect{4,5}"
   Circle "Circle_34" at 301,180 size 27x27
      Appearance <- "Jugador2Vect_J2Vect{4,6}"
   Circle "Circle_35" at 328,180 size 27x27
      Appearance <- "Jugador2Vect_J2Vect{4,7}"
   Circle "Circle_36" at 355,180 size 27x27
      Appearance <- "Jugador2Vect_J2Vect{4,8}"
   Circle "Circle_37" at 139,207 size 27x27
      Appearance <- "Jugador2Vect_J2Vect{3,0}"
   Circle "Circle_38" at 166,207 size 27x27
      Appearance <- "Jugador2Vect_J2Vect{3,1}"
   Circle "Circle_39" at 193,207 size 27x27
      Appearance <- "Jugador2Vect_J2Vect{3,2}"
   Circle "Circle_40" at 220,207 size 27x27
      Appearance <- "Jugador2Vect_J2Vect{3,3}"
   Circle "Circle_41" at 247,207 size 27x27
      Appearance <- "Jugador2Vect_J2Vect{3,4}"
   Circle "Circle_42" at 274,207 size 27x27
      Appearance <- "Jugador2Vect_J2Vect{3,5}"
   Circle "Circle_43" at 301,207 size 27x27
      Appearance <- "Jugador2Vect_J2Vect{3,6}"
   Circle "Circle_44" at 328,207 size 27x27
      Appearance <- "Jugador2Vect_J2Vect{3,7}"
   Circle "Circle_45" at 355,207 size 27x27
      Appearance <- "Jugador2Vect_J2Vect{3,8}"
   Circle "Circle_46" at 139,234 size 27x27
      Appearance <- "Jugador2Vect_J2Vect{2,0}"
   Circle "Circle_47" at 166,234 size 27x27
      Appearance <- "Jugador2Vect_J2Vect{2,1}"
   Circle "Circle_48" at 193,234 size 27x27
      Appearance <- "Jugador2Vect_J2Vect{2,2}"
   Circle "Circle_49" at 220,234 size 27x27
      Appearance <- "Jugador2Vect_J2Vect{2,3}"
   Circle "Circle_50" at 247,234 size 27x27
      Appearance <- "Jugador2Vect_J2Vect{2,4}"
   Circle "Circle_51" at 274,234 size 27x27
      Appearance <- "Jugador2Vect_J2Vect{2,5}"
   Circle "Circle_52" at 301,234 size 27x27
      Appearance <- "Jugador2Vect_J2Vect{2,6}"
   Circle "Circle_53" at 328,234 size 27x27
      Appearance <- "Jugador2Vect_J2Vect{2,7}"
   Circle "Circle_54" at 355,234 size 27x27
      Appearance <- "Jugador2Vect_J2Vect{2,8}"
   Circle "Circle_55" at 139,261 size 27x27
      Appearance <- "Jugador2Vect_J2Vect{1,0}"
   Circle "Circle_56" at 166,261 size 27x27
      Appearance <- "Jugador2Vect_J2Vect{1,1}"
   Circle "Circle_57" at 193,261 size 27x27
      Appearance <- "Jugador2Vect_J2Vect{1,2}"
   Circle "Circle_58" at 220,261 size 27x27
      Appearance <- "Jugador2Vect_J2Vect{1,3}"
   Circle "Circle_59" at 247,261 size 27x27
      Appearance <- "Jugador2Vect_J2Vect{1,4}"
   Circle "Circle_60" at 274,261 size 27x27
      Appearance <- "Jugador2Vect_J2Vect{1,5}"
   Circle "Circle_61" at 301,261 size 27x27
      Appearance <- "Jugador2Vect_J2Vect{1,6}"
   Circle "Circle_62" at 328,261 size 27x27
      Appearance <- "Jugador2Vect_J2Vect{1,7}"
   Circle "Circle_63" at 355,261 size 27x27
      Appearance <- "Jugador2Vect_J2Vect{1,8}"
   Circle "Circle_73" at 139,288 size 27x27
      Appearance <- "Jugador2Vect_J2Vect{0,0}"
   Circle "Circle_74" at 166,288 size 27x27
      Appearance <- "Jugador2Vect_J2Vect{0,1}"
   Circle "Circle_75" at 193,288 size 27x27
      Appearance <- "Jugador2Vect_J2Vect{0,2}"
   Circle "Circle_76" at 220,288 size 27x27
      Appearance <- "Jugador2Vect_J2Vect{0,3}"
   Circle "Circle_77" at 247,288 size 27x27
      Appearance <- "Jugador2Vect_J2Vect{0,4}"
   Circle "Circle_78" at 274,288 size 27x27
      Appearance <- "Jugador2Vect_J2Vect{0,5}"
   Circle "Circle_79" at 301,288 size 27x27
      Appearance <- "Jugador2Vect_J2Vect{0,6}"
   Circle "Circle_80" at 328,288 size 27x27
      Appearance <- "Jugador2Vect_J2Vect{0,7}"
   Circle "Circle_81" at 355,288 size 27x27
      Appearance <- "Jugador2Vect_J2Vect{0,8}"
   TextField "Text field_9" at 11,25 size 111x61; Text 'JUGADOR 2 FICHAS AMARILLAS'
   TextField "Text field_2" at 481,55 size 264x23; Text 'Modo de Juego Seleccionado'
      Visibility <- "Mensaje1J2"

Template "Template_1" 800x420
   Button "Exit" at 720,360 size 78x58; TextOff 'Exit'; PictureOff "ExitRuntime_TP700_Comfort_TR"; PictureOn "ExitRuntime_TP700_Comfort_TR"
      on Release: StopRuntime(0)
   Button "Template_Button" at 640,360 size 78x58; TextOff 'Text'
   Button "Template_Button_1" at 560,360 size 78x58; TextOff 'Text'
   Button "Template_Button_2" at 480,360 size 78x58; TextOff 'Text'
   Button "Template_Button_3" at 400,360 size 78x58; TextOff 'Text'
   Button "Template_Button_4" at 321,360 size 78x58; TextOff 'Text'
   Button "Template_Button_5" at 241,360 size 78x58; TextOff 'Text'
   Button "Template_Button_6" at 161,360 size 78x58; TextOff 'Text'
   Button "Alarms" at 81,360 size 78x58; TextOff 'Alarms'; PictureOff "AlarmDisplay_TP700_Comfort_TR"; PictureOn "AlarmDisplay_TP700_Comfort_TR"
      on Release: function_ef3f5d25("Alarm window_Unacknowledged", -1)
   Button "Start screen" at 1,360 size 78x58; TextOff 'Start screen'; PictureOff "NavigateHome_TP700_Comfort_TR"; PictureOn "NavigateHome_TP700_Comfort_TR"
      on Release: ActivateScreen("Root screen", 0)
*)